# B&R Automation Studio project GAT (part 2)

### CutCamAut.axisfeature - 5PPC2200_AL14_000/mappMotion/CrossCutter/CutCamAut.axisfeature
```
Element CutterCamAutomat (Type=axisfeature)
  Type = CamAutomat
    CamAutomatType = ACOPOS
      CommonParameters:
        Master:
          ValueSource = SetPosition
            AxisReference = gAxisAppAxis_1
            MaxVelocity = 1000
          StartPosition = 0
          StartInterval = SpecifyValue
            Interval = 100
        AdvancedParameters:
          StartStateParameters:
            StartState = 0
            RelMasterStartPos = 0.0
          AdditiveAxes:
            AdditiveMasterValueSource = NotUsed
            AdditiveSlaveValueSource = NotUsed
          MasterStartPositionMode = NotEvaluatedAnew
          ControlSettings:
            CrossLeftBoundary = PositionLimitedHorizontal
            CamChangeImmediately = CurrentMasterMoveDir
          MessageSettings:
            ErrorsInStandby = NoErrorMessages
          TriggerAndLatch:
            Trigger1Delay = 0.0
            Trigger2Delay = 0.0
            SlaveLatchParID = 0
          EventParIDs
          StartIntervals
          Factors:
            SlaveFactorParID = 0
      States:
        State0 = Used
          Events:
            Event[0]:
              Type = MasterStartPosition
              Transition = Immediately
              SynchronousUpdate = Used
              NextState = 1
        State[1]  // Execute first cut
          Cam = Predefined
            PredefinedCam = OneToOne
          MasterFactor = 2000
          SlaveFactor = 2000
          CompensationMode = DistancesBetweenExitEntryPoints
            MasterDistance = 50
            SlaveDistance = 170
            AdvancedParameters = NotUsed
          AdvancedParameters:
            RepeatCounterInit = 0
            MasterValueSource = CommonMaster
          Events:
            Event[0]  // Stop cutting after next cut
              Type = Signal1FromPLC
              Transition = EndOfState
              SynchronousUpdate = Used
              NextState = 3
            Event[1]:
              Type = StateEnd
              Transition = EndOfState
              SynchronousUpdate = Used
              NextState = 2
        State[2]  // Execute cuts
          Cam = Predefined
            PredefinedCam = OneToOne
          MasterFactor = 2000
          SlaveFactor = 2000
          CompensationMode = DistancesBetweenCamCenterPoints
            MasterDistance = 100
            SlaveDistance = 360
            AdvancedParameters = NotUsed
          AdvancedParameters:
            RepeatCounterInit = 0
            MasterValueSource = CommonMaster
          Events:
            Event[0]  // Stop cutting after next cut
              Type = Signal1FromPLC
              Transition = EndOfState
              SynchronousUpdate = Used
              NextState = 3
            Event[1]:
              Type = StateEnd
              Transition = EndOfState
              SynchronousUpdate = Used
              NextState = 2
        State[3]  // decelerate and stop at home position
          Cam = Predefined
            PredefinedCam = ZeroPoint
          MasterFactor = 1000
          SlaveFactor = 0
          CompensationMode = DistancesBetweenCamCenterPoints
            MasterDistance = 50
            SlaveDistance = 180
            AdvancedParameters = NotUsed
          AdvancedParameters:
            RepeatCounterInit = 0
            MasterValueSource = CommonMaster
          Events:
            Event[0]:
              Type = StateEnd
              Transition = EndOfState
              SynchronousUpdate = Used
              NextState = 0
```

### CutVirt.purevaxcfg - 5PPC2200_AL14_000/mappMotion/CrossCutter/CutVirt.purevaxcfg
```
Element PureVAxCfg_CrossCutter (Type=purevaxcfg)
  TypeID = PureVAxConfig
  PureVAxis:
    AxisReference = gAxisCrossCutter
    Homing:
      Mode = Direct
        Position = 0.0
        ReferencePulse = NotUsed
      RestorePositionVariable
    JerkFilter = NotUsed
    AxisFeatures:
      FeatureRef[1] = CutterCamAutomat
```

### Alarm.mpalarmxcore - 5PPC2200_AL14_000/mappServices/AlarmX/Alarm.mpalarmxcore
```
Element gAlarmXMpLink (Type=mpalarmxcore)
  mapp.AlarmX.Core:
    BySeverity:
      [0]:
        Severity = 1..9
        [0] = Reaction
          Name = Info
      [1]:
        Severity = 10..19
        [0] = Reaction
          Name = Warning
      [2]:
        Severity = 20..29
        [0] = Reaction
          Name = Error
  mapp.AlarmX.Core.Configuration:
    [0]:
      Name = EmergencyStop_0
      Message = {$Alarms/EmergencyStop.0}
      Severity = 29
      Behavior = DiscreteValueMonitoring
        Monitoring:
          MonitoredPV = ::AlarmMgt:SafetyInputs.EmergencyStop[0]
          TriggerValues:
            [0] = 1
    [1]:
      Name = EmergencyStop_1
      Message = {$Alarms/EmergencyStop.1}
      Behavior = DiscreteValueMonitoring
        Monitoring:
          MonitoredPV = ::AlarmMgt:SafetyInputs.EmergencyStop[1]
          TriggerValues:
            [0] = 1
    [2]:
      Name = EmergencyStop_2
      Message = {$Alarms/EmergencyStop.2}
      Behavior = DiscreteValueMonitoring
        Monitoring:
          MonitoredPV = ::AlarmMgt:SafetyInputs.EmergencyStop[2]
          TriggerValues:
            [0] = 1
    [3]:
      Name = SafetyDoor_0
      Message = {$Alarms/SafetyDoor.0}
      Severity = 29
      Behavior = DiscreteValueMonitoring
        Monitoring:
          MonitoredPV = ::AlarmMgt:SafetyInputs.SafetyDoor[0]
          TriggerValues:
            [0] = 1
    [4]:
      Name = SafetyDoor_1
      Message = {$Alarms/SafetyDoor.1}
      Severity = 29
      Behavior = DiscreteValueMonitoring
        Monitoring:
          MonitoredPV = ::AlarmMgt:SafetyInputs.SafetyDoor[1]
          TriggerValues:
            [0] = 1
    [5]:
      Name = SafetyDoor_2
      Message = {$Alarms/SafetyDoor.2}
      Severity = 29
      Behavior = DiscreteValueMonitoring
        Monitoring:
          MonitoredPV = ::AlarmMgt:SafetyInputs.SafetyDoor[2]
          TriggerValues:
            [0] = 1
    [6]:
      Name = SafetyDoor_3
      Message = {$Alarms/SafetyDoor.3}
      Severity = 29
      Behavior = DiscreteValueMonitoring
        Monitoring:
          MonitoredPV = ::AlarmMgt:SafetyInputs.SafetyDoor[3]
          TriggerValues:
            [0] = 1
    [7]:
      Name = SafetyDoor_4
      Message = {$Alarms/SafetyDoor.4}
      Severity = 29
      Behavior = DiscreteValueMonitoring
        Monitoring:
          MonitoredPV = ::AlarmMgt:SafetyInputs.SafetyDoor[4]
          TriggerValues:
            [0] = 1
    [8]:
      Name = SafetyDoor_5
      Message = {$Alarms/SafetyDoor.5}
      Severity = 29
      Behavior = DiscreteValueMonitoring
        Monitoring:
          MonitoredPV = ::AlarmMgt:SafetyInputs.SafetyDoor[5]
          TriggerValues:
            [0] = 1
    [9]:
      Name = LevelMonitoringExample
      Message = {$Alarms/LevelMonitoringAlarmExample} {=$Alarms/{&LimitText}}
      Behavior = LevelMonitoring
        Monitoring:
          MonitoredPV = ::AlarmMgt:AlarmExamples.LevelMonitoring
          LowLimitEnable = Static
            Limit = 20
            LimitText = LevelMonitoringAlarmLowTextExample
            LowLowLimitEnable = Static
              Limit = 10
              LimitText = LevelMonitoringAlarmLowLowTextExample
          HighLimitEnable = Static
            Limit = 80
            LimitText = LevelMonitoringAlarmHighTextExample
            HighHighLimitEnable = Static
              Limit = 90
              LimitText = LevelMonitoringAlarmHighHighTextExample
    [10]:
      Name = DeviationMonitoringExample
      Message = {$Alarms/DeviationMonitoringAlarmExample} {&LimitText}
      Behavior = DeviationMonitoring
        Monitoring:
          MonitoredPV = ::AlarmMgt:AlarmExamples.DeviationMonitoring
          SetpointPV = ::AlarmMgt:AlarmExamples.DeviationMonitoringSetpoint
          LowLimitEnable = Static
            Limit = -5
            LimitText = Low limit exceeded
          HighLimitEnable = Static
            Limit = 5
            LimitText = High limit exceeded
    [11]:
      Name = RateOfChangeExample
      Message = {$Alarms/RateOfChangeAlarmExample}
      Behavior = RateOfChangeMonitoring
        Monitoring:
          MonitoredPV = ::AlarmMgt:AlarmExamples.RateOfChange
          HighLimitEnable = Static
            Limit = 5
            LimitText = High limit exceeded
    [12]:
      Name = SnippetExample
      Message = Show a snippet: {&snippet1}
      Behavior = DiscreteValueMonitoring
        Monitoring:
          MonitoredPV = ::AlarmMgt:AlarmExamples.SnippetValue
          TriggerValues:
            [0] = 50..100
    [13]:
      Name = MpAlarmXControlExample
      Message = {$Alarms/MpAlarmXControlExample}
      Severity = 20
      Behavior:
        Async = TRUE
    [14]:
      Name = Alarm0
      Message = {$Alarms/Alarm.0}
      Behavior = DiscreteValueMonitoring
        Monitoring:
          MonitoredPV = ::AlarmMgt:Alarms[0]
          InhibitPV = ::AlarmMgt:CommissioningModeActive
          TriggerValues:
            [0] = 1
    [15]:
      Name = Alarm1
      Message = {$Alarms/Alarm.1}
      Code = 1
      Behavior = DiscreteValueMonitoring
        Monitoring:
          MonitoredPV = ::AlarmMgt:Alarms[1]
          TriggerValues:
            [0] = 1
    [16]:
      Name = Alarm2
      Message = {$Alarms/Alarm.2}
      Code = 2
      Behavior = DiscreteValueMonitoring
        Monitoring:
          MonitoredPV = ::AlarmMgt:Alarms[2]
          TriggerValues:
            [0] = 1
    [17]:
      Name = Alarm3
      Message = {$Alarms/Alarm.3}
      Code = 3
      Behavior = DiscreteValueMonitoring
        Monitoring:
          MonitoredPV = ::AlarmMgt:Alarms[3]
          TriggerValues:
            [0] = 1
    [18]:
      Name = Alarm4
      Message = {$Alarms/Alarm.4}
      Code = 4
      Behavior = DiscreteValueMonitoring
        Monitoring:
          MonitoredPV = ::AlarmMgt:Alarms[4]
          TriggerValues:
            [0] = 1
    [19]:
      Name = Alarm5
      Message = {$Alarms/Alarm.5}
      Code = 5
      Behavior = DiscreteValueMonitoring
        Monitoring:
          MonitoredPV = ::AlarmMgt:Alarms[5]
          TriggerValues:
            [0] = 1
    [20]:
      Name = Alarm6
      Message = {$Alarms/Alarm.6}
      Code = 6
      Behavior = DiscreteValueMonitoring
        Monitoring:
          MonitoredPV = ::AlarmMgt:Alarms[6]
          TriggerValues:
            [0] = 1
    [21]:
      Name = Alarm7
      Message = {$Alarms/Alarm.7}
      Code = 7
      Behavior = DiscreteValueMonitoring
        Monitoring:
          MonitoredPV = ::AlarmMgt:Alarms[7]
          TriggerValues:
            [0] = 1
    [22]:
      Name = Alarm8
      Message = {$Alarms/Alarm.8}
      Code = 8
      Behavior = DiscreteValueMonitoring
        Monitoring:
          MonitoredPV = ::AlarmMgt:Alarms[8]
          TriggerValues:
            [0] = 1
    [23]:
      Name = Alarm9
      Message = {$Alarms/Alarm.9}
      Code = 9
      Behavior = DiscreteValueMonitoring
        Monitoring:
          MonitoredPV = ::AlarmMgt:Alarms[9]
          TriggerValues:
            [0] = 1
    [24]:
      Name = Alarm10
      Message = {$Alarms/Alarm.10}
      Code = 10
      Behavior = DiscreteValueMonitoring
        Monitoring:
          MonitoredPV = ::AlarmMgt:Alarms[10]
          TriggerValues:
            [0] = 1
    [25]:
      Name = Alarm11
      Message = {$Alarms/Alarm.11}
      Code = 11
      Behavior = DiscreteValueMonitoring
        Monitoring:
          MonitoredPV = ::AlarmMgt:Alarms[11]
          TriggerValues:
            [0] = 1
    [26]:
      Name = Alarm12
      Message = {$Alarms/Alarm.12}
      Code = 12
      Behavior = DiscreteValueMonitoring
        Monitoring:
          MonitoredPV = ::AlarmMgt:Alarms[12]
          TriggerValues:
            [0] = 1
    [27]:
      Name = Alarm13
      Message = {$Alarms/Alarm.13}
      Code = 13
      Behavior = DiscreteValueMonitoring
        Monitoring:
          MonitoredPV = ::AlarmMgt:Alarms[13]
          TriggerValues:
            [0] = 1
    [28]:
      Name = Alarm14
      Message = {$Alarms/Alarm.14}
      Code = 14
      Behavior = DiscreteValueMonitoring
        Monitoring:
          MonitoredPV = ::AlarmMgt:Alarms[14]
          TriggerValues:
            [0] = 1
    [29]:
      Name = Alarm15
      Message = {$Alarms/Alarm.15}
      Code = 15
      Behavior = DiscreteValueMonitoring
        Monitoring:
          MonitoredPV = ::AlarmMgt:Alarms[15]
          TriggerValues:
            [0] = 1
    [30]:
      Name = Alarm16
      Message = {$Alarms/Alarm.16}
      Code = 16
      Behavior = DiscreteValueMonitoring
        Monitoring:
          MonitoredPV = ::AlarmMgt:Alarms[16]
          TriggerValues:
            [0] = 1
    [31]:
      Name = Alarm17
      Message = {$Alarms/Alarm.17}
      Code = 17
      Behavior = DiscreteValueMonitoring
        Monitoring:
          MonitoredPV = ::AlarmMgt:Alarms[17]
          TriggerValues:
            [0] = 1
    [32]:
      Name = Alarm18
      Message = {$Alarms/Alarm.18}
      Code = 18
      Behavior = DiscreteValueMonitoring
        Monitoring:
          MonitoredPV = ::AlarmMgt:Alarms[18]
          TriggerValues:
            [0] = 1
    [33]:
      Name = Alarm19
      Message = {$Alarms/Alarm.19}
      Code = 19
      Behavior = DiscreteValueMonitoring
        Monitoring:
          MonitoredPV = ::AlarmMgt:Alarms[19]
          TriggerValues:
            [0] = 1
    [34]:
      Name = Alarm20
      Message = {$Alarms/Alarm.20}
      Behavior = DiscreteValueMonitoring
        Monitoring:
          MonitoredPV = ::AlarmMgt:Alarms[20]
          TriggerValues:
            [0] = 1
    [35]:
      Name = Alarm21
      Message = {$Alarms/Alarm.21}
      Code = 21
      Behavior = DiscreteValueMonitoring
        Monitoring:
          MonitoredPV = ::AlarmMgt:Alarms[21]
          TriggerValues:
            [0] = 1
    [36]:
      Name = Alarm22
      Message = {$Alarms/Alarm.22}
      Code = 22
      Behavior = DiscreteValueMonitoring
        Monitoring:
          MonitoredPV = ::AlarmMgt:Alarms[22]
          TriggerValues:
            [0] = 1
    [37]:
      Name = Alarm23
      Message = {$Alarms/Alarm.23}
      Code = 23
      Behavior = DiscreteValueMonitoring
        Monitoring:
          MonitoredPV = ::AlarmMgt:Alarms[23]
          TriggerValues:
            [0] = 1
    [38]:
      Name = Alarm24
      Message = {$Alarms/Alarm.24}
      Code = 24
      Behavior = DiscreteValueMonitoring
        Monitoring:
          MonitoredPV = ::AlarmMgt:Alarms[24]
          TriggerValues:
            [0] = 1
    [39]:
      Name = Alarm25
      Message = {$Alarms/Alarm.25}
      Code = 25
      Behavior = DiscreteValueMonitoring
        Monitoring:
          MonitoredPV = ::AlarmMgt:Alarms[25]
          TriggerValues:
            [0] = 1
    [40]:
      Name = Alarm26
      Message = {$Alarms/Alarm.26}
      Code = 26
      Behavior = DiscreteValueMonitoring
        Monitoring:
          MonitoredPV = ::AlarmMgt:Alarms[26]
          TriggerValues:
            [0] = 1
    [41]:
      Name = Alarm27
      Message = {$Alarms/Alarm.27}
      Code = 27
      Behavior = DiscreteValueMonitoring
        Monitoring:
          MonitoredPV = ::AlarmMgt:Alarms[27]
          TriggerValues:
            [0] = 1
    [42]:
      Name = Alarm28
      Message = {$Alarms/Alarm.28}
      Code = 28
      Behavior = DiscreteValueMonitoring
        Monitoring:
          MonitoredPV = ::AlarmMgt:Alarms[28]
          TriggerValues:
            [0] = 1
    [43]:
      Name = Alarm29
      Message = {$Alarms/Alarm.29}
      Code = 29
      Behavior = DiscreteValueMonitoring
        Monitoring:
          MonitoredPV = ::AlarmMgt:Alarms[29]
          TriggerValues:
            [0] = 1
    [44]:
      Name = Alarm30
      Message = {$Alarms/Alarm.30}
      Behavior = DiscreteValueMonitoring
        Monitoring:
          MonitoredPV = ::AlarmMgt:Alarms[30]
          TriggerValues:
            [0] = 1
    [45]:
      Name = Alarm31
      Message = {$Alarms/Alarm.31}
      Code = 31
      Behavior = DiscreteValueMonitoring
        Monitoring:
          MonitoredPV = ::AlarmMgt:Alarms[31]
          TriggerValues:
            [0] = 1
    [46]:
      Name = Alarm32
      Message = {$Alarms/Alarm.32}
      Code = 32
      Behavior = DiscreteValueMonitoring
        Monitoring:
          MonitoredPV = ::AlarmMgt:Alarms[32]
          TriggerValues:
            [0] = 1
    [47]:
      Name = Alarm33
      Message = {$Alarms/Alarm.33}
      Code = 33
      Behavior = DiscreteValueMonitoring
        Monitoring:
          MonitoredPV = ::AlarmMgt:Alarms[33]
          TriggerValues:
            [0] = 1
    [48]:
      Name = Alarm34
      Message = {$Alarms/Alarm.34}
      Code = 34
      Behavior = DiscreteValueMonitoring
        Monitoring:
          MonitoredPV = ::AlarmMgt:Alarms[34]
          TriggerValues:
            [0] = 1
    [49]:
      Name = Alarm35
      Message = {$Alarms/Alarm.35}
      Code = 35
      Behavior = DiscreteValueMonitoring
        Monitoring:
          MonitoredPV = ::AlarmMgt:Alarms[35]
          TriggerValues:
            [0] = 1
    [50]:
      Name = Alarm36
      Message = {$Alarms/Alarm.36}
      Code = 36
      Behavior = DiscreteValueMonitoring
        Monitoring:
          MonitoredPV = ::AlarmMgt:Alarms[36]
          TriggerValues:
            [0] = 1
    [51]:
      Name = Alarm37
      Message = {$Alarms/Alarm.37}
      Code = 37
      Behavior = DiscreteValueMonitoring
        Monitoring:
          MonitoredPV = ::AlarmMgt:Alarms[37]
          TriggerValues:
            [0] = 1
    [52]:
      Name = Alarm38
      Message = {$Alarms/Alarm.38}
      Code = 38
      Behavior = DiscreteValueMonitoring
        Monitoring:
          MonitoredPV = ::AlarmMgt:Alarms[38]
          TriggerValues:
            [0] = 1
    [53]:
      Name = Alarm39
      Message = {$Alarms/Alarm.39}
      Code = 39
      Behavior = DiscreteValueMonitoring
        Monitoring:
          MonitoredPV = ::AlarmMgt:Alarms[39]
          TriggerValues:
            [0] = 1
    [54]:
      Name = Alarm40
      Message = {$Alarms/Alarm.40}
      Behavior = DiscreteValueMonitoring
        Monitoring:
          MonitoredPV = ::AlarmMgt:Alarms[40]
          TriggerValues:
            [0] = 1
    [55]:
      Name = Alarm41
      Message = {$Alarms/Alarm.41}
      Code = 41
      Behavior = DiscreteValueMonitoring
        Monitoring:
          MonitoredPV = ::AlarmMgt:Alarms[41]
          TriggerValues:
            [0] = 1
    [56]:
      Name = Alarm42
      Message = {$Alarms/Alarm.42}
      Code = 42
      Behavior = DiscreteValueMonitoring
        Monitoring:
          MonitoredPV = ::AlarmMgt:Alarms[42]
          TriggerValues:
            [0] = 1
    [57]:
      Name = Alarm43
      Message = {$Alarms/Alarm.43}
      Code = 43
      Behavior = DiscreteValueMonitoring
        Monitoring:
          MonitoredPV = ::AlarmMgt:Alarms[43]
          TriggerValues:
            [0] = 1
    [58]:
      Name = Alarm44
      Message = {$Alarms/Alarm.44}
      Code = 44
      Behavior = DiscreteValueMonitoring
        Monitoring:
          MonitoredPV = ::AlarmMgt:Alarms[44]
          TriggerValues:
            [0] = 1
    [59]:
      Name = Alarm45
      Message = {$Alarms/Alarm.45}
      Code = 45
      Behavior = DiscreteValueMonitoring
        Monitoring:
          MonitoredPV = ::AlarmMgt:Alarms[45]
          TriggerValues:
            [0] = 1
    [60]:
      Name = Alarm46
      Message = {$Alarms/Alarm.46}
      Code = 46
      Behavior = DiscreteValueMonitoring
        Monitoring:
          MonitoredPV = ::AlarmMgt:Alarms[46]
          TriggerValues:
            [0] = 1
    [61]:
      Name = Alarm47
      Message = {$Alarms/Alarm.47}
      Code = 47
      Behavior = DiscreteValueMonitoring
        Monitoring:
          MonitoredPV = ::AlarmMgt:Alarms[47]
          TriggerValues:
            [0] = 1
    [62]:
      Name = Alarm48
      Message = {$Alarms/Alarm.48}
      Code = 48
      Behavior = DiscreteValueMonitoring
        Monitoring:
          MonitoredPV = ::AlarmMgt:Alarms[48]
          TriggerValues:
            [0] = 1
    [63]:
      Name = Alarm49
      Message = {$Alarms/Alarm.49}
      Code = 49
      Behavior = DiscreteValueMonitoring
        Monitoring:
          MonitoredPV = ::AlarmMgt:Alarms[49]
          TriggerValues:
            [0] = 1
    [64]:
      Name = Alarm50
      Message = {$Alarms/Alarm.50}
      Behavior = DiscreteValueMonitoring
        Monitoring:
          MonitoredPV = ::AlarmMgt:Alarms[50]
          TriggerValues:
            [0] = 1
    [65]:
      Name = Alarm51
      Message = {$Alarms/Alarm.51}
      Code = 51
      Behavior = DiscreteValueMonitoring
        Monitoring:
          MonitoredPV = ::AlarmMgt:Alarms[51]
          TriggerValues:
            [0] = 1
    [66]:
      Name = Alarm52
      Message = {$Alarms/Alarm.52}
      Code = 52
      Behavior = DiscreteValueMonitoring
        Monitoring:
          MonitoredPV = ::AlarmMgt:Alarms[52]
          TriggerValues:
            [0] = 1
    [67]:
      Name = Alarm53
      Message = {$Alarms/Alarm.53}
      Code = 53
      Behavior = DiscreteValueMonitoring
        Monitoring:
          MonitoredPV = ::AlarmMgt:Alarms[53]
          TriggerValues:
            [0] = 1
    [68]:
      Name = Alarm54
      Message = {$Alarms/Alarm.54}
      Code = 54
      Behavior = DiscreteValueMonitoring
        Monitoring:
          MonitoredPV = ::AlarmMgt:Alarms[54]
          TriggerValues:
            [0] = 1
    [69]:
      Name = Alarm55
      Message = {$Alarms/Alarm.55}
      Code = 55
      Behavior = DiscreteValueMonitoring
        Monitoring:
          MonitoredPV = ::AlarmMgt:Alarms[55]
          TriggerValues:
            [0] = 1
    [70]:
      Name = Alarm56
      Message = {$Alarms/Alarm.56}
      Code = 56
      Behavior = DiscreteValueMonitoring
        Monitoring:
          MonitoredPV = ::AlarmMgt:Alarms[56]
          TriggerValues:
            [0] = 1
    [71]:
      Name = Alarm57
      Message = {$Alarms/Alarm.57}
      Code = 57
      Behavior = DiscreteValueMonitoring
        Monitoring:
          MonitoredPV = ::AlarmMgt:Alarms[57]
          TriggerValues:
            [0] = 1
    [72]:
      Name = Alarm58
      Message = {$Alarms/Alarm.58}
      Code = 58
      Behavior = DiscreteValueMonitoring
        Monitoring:
          MonitoredPV = ::AlarmMgt:Alarms[58]
          TriggerValues:
            [0] = 1
    [73]:
      Name = Alarm59
      Message = {$Alarms/Alarm.59}
      Code = 59
      Behavior = DiscreteValueMonitoring
        Monitoring:
          MonitoredPV = ::AlarmMgt:Alarms[59]
          TriggerValues:
            [0] = 1
    [74]:
      Name = Alarm60
      Message = {$Alarms/Alarm.60}
      Behavior = DiscreteValueMonitoring
        Monitoring:
          MonitoredPV = ::AlarmMgt:Alarms[60]
          TriggerValues:
            [0] = 1
    [75]:
      Name = Alarm61
      Message = {$Alarms/Alarm.61}
      Code = 61
      Behavior = DiscreteValueMonitoring
        Monitoring:
          MonitoredPV = ::AlarmMgt:Alarms[61]
          TriggerValues:
            [0] = 1
    [76]:
      Name = Alarm62
      Message = {$Alarms/Alarm.62}
      Code = 62
      Behavior = DiscreteValueMonitoring
        Monitoring:
          MonitoredPV = ::AlarmMgt:Alarms[62]
          TriggerValues:
            [0] = 1
    [77]:
      Name = Alarm63
      Message = {$Alarms/Alarm.63}
      Code = 63
      Behavior = DiscreteValueMonitoring
        Monitoring:
          MonitoredPV = ::AlarmMgt:Alarms[63]
          TriggerValues:
            [0] = 1
    [78]:
      Name = Alarm64
      Message = {$Alarms/Alarm.64}
      Code = 64
      Behavior = DiscreteValueMonitoring
        Monitoring:
          MonitoredPV = ::AlarmMgt:Alarms[64]
          TriggerValues:
            [0] = 1
    [79]:
      Name = Alarm65
      Message = {$Alarms/Alarm.65}
      Code = 65
      Behavior = DiscreteValueMonitoring
        Monitoring:
          MonitoredPV = ::AlarmMgt:Alarms[65]
          TriggerValues:
            [0] = 1
    [80]:
      Name = Alarm66
      Message = {$Alarms/Alarm.66}
      Code = 66
      Behavior = DiscreteValueMonitoring
        Monitoring:
          MonitoredPV = ::AlarmMgt:Alarms[66]
          TriggerValues:
            [0] = 1
    [81]:
      Name = Alarm67
      Message = {$Alarms/Alarm.67}
      Code = 67
      Behavior = DiscreteValueMonitoring
        Monitoring:
          MonitoredPV = ::AlarmMgt:Alarms[67]
          TriggerValues:
            [0] = 1
    [82]:
      Name = Alarm68
      Message = {$Alarms/Alarm.68}
      Code = 68
      Behavior = DiscreteValueMonitoring
        Monitoring:
          MonitoredPV = ::AlarmMgt:Alarms[68]
          TriggerValues:
            [0] = 1
    [83]:
      Name = Alarm69
      Message = {$Alarms/Alarm.69}
      Code = 69
      Behavior = DiscreteValueMonitoring
        Monitoring:
          MonitoredPV = ::AlarmMgt:Alarms[69]
          TriggerValues:
            [0] = 1
    [84]:
      Name = Alarm70
      Message = {$Alarms/Alarm.70}
      Behavior = DiscreteValueMonitoring
        Monitoring:
          MonitoredPV = ::AlarmMgt:Alarms[70]
          TriggerValues:
            [0] = 1
    [85]:
      Name = Alarm71
      Message = {$Alarms/Alarm.71}
      Code = 71
      Behavior = DiscreteValueMonitoring
        Monitoring:
          MonitoredPV = ::AlarmMgt:Alarms[71]
          TriggerValues:
            [0] = 1
    [86]:
      Name = Alarm72
      Message = {$Alarms/Alarm.72}
      Code = 72
      Behavior = DiscreteValueMonitoring
        Monitoring:
          MonitoredPV = ::AlarmMgt:Alarms[72]
          TriggerValues:
            [0] = 1
    [87]:
      Name = Alarm73
      Message = {$Alarms/Alarm.73}
      Code = 73
      Behavior = DiscreteValueMonitoring
        Monitoring:
          MonitoredPV = ::AlarmMgt:Alarms[73]
          TriggerValues:
            [0] = 1
    [88]:
      Name = Alarm74
      Message = {$Alarms/Alarm.74}
      Code = 74
      Behavior = DiscreteValueMonitoring
        Monitoring:
          MonitoredPV = ::AlarmMgt:Alarms[74]
          TriggerValues:
            [0] = 1
    [89]:
      Name = Alarm75
      Message = {$Alarms/Alarm.75}
      Code = 75
      Behavior = DiscreteValueMonitoring
        Monitoring:
          MonitoredPV = ::AlarmMgt:Alarms[75]
          TriggerValues:
            [0] = 1
    [90]:
      Name = Alarm76
      Message = {$Alarms/Alarm.76}
      Code = 76
      Behavior = DiscreteValueMonitoring
        Monitoring:
          MonitoredPV = ::AlarmMgt:Alarms[76]
          TriggerValues:
            [0] = 1
    [91]:
      Name = Alarm77
      Message = {$Alarms/Alarm.77}
      Code = 77
      Behavior = DiscreteValueMonitoring
        Monitoring:
          MonitoredPV = ::AlarmMgt:Alarms[77]
          TriggerValues:
            [0] = 1
    [92]:
      Name = Alarm78
      Message = {$Alarms/Alarm.78}
      Code = 78
      Behavior = DiscreteValueMonitoring
        Monitoring:
          MonitoredPV = ::AlarmMgt:Alarms[78]
          TriggerValues:
            [0] = 1
    [93]:
      Name = Alarm79
      Message = {$Alarms/Alarm.79}
      Code = 79
      Behavior = DiscreteValueMonitoring
        Monitoring:
          MonitoredPV = ::AlarmMgt:Alarms[79]
          TriggerValues:
            [0] = 1
    [94]:
      Name = Alarm80
      Message = {$Alarms/Alarm.80}
      Behavior = DiscreteValueMonitoring
        Monitoring:
          MonitoredPV = ::AlarmMgt:Alarms[80]
          TriggerValues:
            [0] = 1
    [95]:
      Name = Alarm81
      Message = {$Alarms/Alarm.81}
      Code = 81
      Behavior = DiscreteValueMonitoring
        Monitoring:
          MonitoredPV = ::AlarmMgt:Alarms[81]
          TriggerValues:
            [0] = 1
    [96]:
      Name = Alarm82
      Message = {$Alarms/Alarm.82}
      Code = 82
      Behavior = DiscreteValueMonitoring
        Monitoring:
          MonitoredPV = ::AlarmMgt:Alarms[82]
          TriggerValues:
            [0] = 1
    [97]:
      Name = Alarm83
      Message = {$Alarms/Alarm.83}
      Code = 83
      Behavior = DiscreteValueMonitoring
        Monitoring:
          MonitoredPV = ::AlarmMgt:Alarms[83]
          TriggerValues:
            [0] = 1
    [98]:
      Name = Alarm84
      Message = {$Alarms/Alarm.84}
      Code = 84
      Behavior = DiscreteValueMonitoring
        Monitoring:
          MonitoredPV = ::AlarmMgt:Alarms[84]
          TriggerValues:
            [0] = 1
    [99]:
      Name = Alarm85
      Message = {$Alarms/Alarm.85}
      Code = 85
      Behavior = DiscreteValueMonitoring
        Monitoring:
          MonitoredPV = ::AlarmMgt:Alarms[85]
          TriggerValues:
            [0] = 1
    [100]:
      Name = Alarm86
      Message = {$Alarms/Alarm.86}
      Code = 86
      Behavior = DiscreteValueMonitoring
        Monitoring:
          MonitoredPV = ::AlarmMgt:Alarms[86]
          TriggerValues:
            [0] = 1
    [101]:
      Name = Alarm87
      Message = {$Alarms/Alarm.87}
      Code = 87
      Behavior = DiscreteValueMonitoring
        Monitoring:
          MonitoredPV = ::AlarmMgt:Alarms[87]
          TriggerValues:
            [0] = 1
    [102]:
      Name = Alarm88
      Message = {$Alarms/Alarm.88}
      Code = 88
      Behavior = DiscreteValueMonitoring
        Monitoring:
          MonitoredPV = ::AlarmMgt:Alarms[88]
          TriggerValues:
            [0] = 1
    [103]:
      Name = Alarm89
      Message = {$Alarms/Alarm.89}
      Code = 89
      Behavior = DiscreteValueMonitoring
        Monitoring:
          MonitoredPV = ::AlarmMgt:Alarms[89]
          TriggerValues:
            [0] = 1
    [104]:
      Name = Alarm90
      Message = {$Alarms/Alarm.90}
      Behavior = DiscreteValueMonitoring
        Monitoring:
          MonitoredPV = ::AlarmMgt:Alarms[90]
          TriggerValues:
            [0] = 1
    [105]:
      Name = Alarm91
      Message = {$Alarms/Alarm.91}
      Code = 91
      Behavior = DiscreteValueMonitoring
        Monitoring:
          MonitoredPV = ::AlarmMgt:Alarms[91]
          TriggerValues:
            [0] = 1
    [106]:
      Name = Alarm92
      Message = {$Alarms/Alarm.92}
      Code = 92
      Behavior = DiscreteValueMonitoring
        Monitoring:
          MonitoredPV = ::AlarmMgt:Alarms[92]
          TriggerValues:
            [0] = 1
    [107]:
      Name = Alarm93
      Message = {$Alarms/Alarm.93}
      Code = 93
      Behavior = DiscreteValueMonitoring
        Monitoring:
          MonitoredPV = ::AlarmMgt:Alarms[93]
          TriggerValues:
            [0] = 1
    [108]:
      Name = Alarm94
      Message = {$Alarms/Alarm.94}
      Code = 94
      Behavior = DiscreteValueMonitoring
        Monitoring:
          MonitoredPV = ::AlarmMgt:Alarms[94]
          TriggerValues:
            [0] = 1
    [109]:
      Name = Alarm95
      Message = {$Alarms/Alarm.95}
      Code = 95
      Behavior = DiscreteValueMonitoring
        Monitoring:
          MonitoredPV = ::AlarmMgt:Alarms[95]
          TriggerValues:
            [0] = 1
    [110]:
      Name = Alarm96
      Message = {$Alarms/Alarm.96}
      Code = 96
      Behavior = DiscreteValueMonitoring
        Monitoring:
          MonitoredPV = ::AlarmMgt:Alarms[96]
          TriggerValues:
            [0] = 1
    [111]:
      Name = Alarm97
      Message = {$Alarms/Alarm.97}
      Code = 97
      Behavior = DiscreteValueMonitoring
        Monitoring:
          MonitoredPV = ::AlarmMgt:Alarms[97]
          TriggerValues:
            [0] = 1
    [112]:
      Name = Alarm98
      Message = {$Alarms/Alarm.98}
      Code = 98
      Behavior = DiscreteValueMonitoring
        Monitoring:
          MonitoredPV = ::AlarmMgt:Alarms[98]
          TriggerValues:
            [0] = 1
    [113]:
      Name = Alarm99
      Message = {$Alarms/Alarm.99}
      Code = 99
      Behavior = DiscreteValueMonitoring
        Monitoring:
          MonitoredPV = ::AlarmMgt:Alarms[99]
          TriggerValues:
            [0] = 1
  mapp.AlarmX.Core.Snippets:
    AutoDetect = 1
    [0]:
      Key = snippet1
      Value:
        PV = ::AlarmMgt:AlarmExamples.SnippetValue
  mapp.AlarmX.Core.Queries:
    [0]:
      Name = ActiveAlarms
      Update = ::AlarmMgt:AlarmQuery.ActiveAlarmUpdateCount
      Source:
        SELECT:
          [0]:
            PV = ::AlarmMgt:AlarmQuery.Alarms[].Name
          [1]:
            Column = Message
            PV = ::AlarmMgt:AlarmQuery.Alarms[].Message
          [2]:
            Column = Code
            PV = ::AlarmMgt:AlarmQuery.Alarms[].Code
          [3]:
            Column = Severity
            PV = ::AlarmMgt:AlarmQuery.Alarms[].Severity
          [4]:
            Column = Scope
            PV = ::AlarmMgt:AlarmQuery.Alarms[].Scope
          [5]:
            Column = TimeStamp
            PV = ::AlarmMgt:AlarmQuery.Alarms[].TimeStamp
          [6]:
            Column = AdditionalInformation1
            PV = ::AlarmMgt:AlarmQuery.Alarms[].AdditionalInfo
          [7]:
            Column = StateActive
            PV = ::AlarmMgt:AlarmQuery.Alarms[].Active
          [8]:
            Column = StateAcknowledged
            PV = ::AlarmMgt:AlarmQuery.Alarms[].Acknowledged
```

### AlarmX.mpalarmxcore - 5PPC2200_AL14_000/mappServices/AlarmX/AlarmX.mpalarmxcore
```
Element gMpLinkAlarmXCore (Type=mpalarmxcore)
  mapp.AlarmX.Core:
    BySeverity:
      [0]:
        Severity = 1..9
        [0] = Reaction
          Name = Info
      [1]:
        Severity = 10..19
        [0] = Reaction
          Name = Warning
      [2]:
        Severity = 20..29
        [0] = Reaction
          Name = Error
  mapp.AlarmX.Core.Configuration:
    [0]:
      Name = EmergencyStop_0
      Message = {$Alarms/EmergencyStop.0}
      Severity = 29
      Behavior = DiscreteValueMonitoring
        Monitoring:
          MonitoredPV = ::AlarmMgt:SafetyInputs.EmergencyStop[0]
          TriggerValues:
            [0] = 1
    [1]:
      Name = EmergencyStop_1
      Message = {$Alarms/EmergencyStop.1}
      Behavior = DiscreteValueMonitoring
        Monitoring:
          MonitoredPV = ::AlarmMgt:SafetyInputs.EmergencyStop[1]
          TriggerValues:
            [0] = 1
    [2]:
      Name = EmergencyStop_2
      Message = {$Alarms/EmergencyStop.2}
      Behavior = DiscreteValueMonitoring
        Monitoring:
          MonitoredPV = ::AlarmMgt:SafetyInputs.EmergencyStop[2]
          TriggerValues:
            [0] = 1
    [3]:
      Name = SafetyDoor_0
      Message = {$Alarms/SafetyDoor.0}
      Severity = 29
      Behavior = DiscreteValueMonitoring
        Monitoring:
          MonitoredPV = ::AlarmMgt:SafetyInputs.SafetyDoor[0]
          TriggerValues:
            [0] = 1
    [4]:
      Name = SafetyDoor_1
      Message = {$Alarms/SafetyDoor.1}
      Severity = 29
      Behavior = DiscreteValueMonitoring
        Monitoring:
          MonitoredPV = ::AlarmMgt:SafetyInputs.SafetyDoor[1]
          TriggerValues:
            [0] = 1
    [5]:
      Name = SafetyDoor_2
      Message = {$Alarms/SafetyDoor.2}
      Severity = 29
      Behavior = DiscreteValueMonitoring
        Monitoring:
          MonitoredPV = ::AlarmMgt:SafetyInputs.SafetyDoor[2]
          TriggerValues:
            [0] = 1
    [6]:
      Name = SafetyDoor_3
      Message = {$Alarms/SafetyDoor.3}
      Severity = 29
      Behavior = DiscreteValueMonitoring
        Monitoring:
          MonitoredPV = ::AlarmMgt:SafetyInputs.SafetyDoor[3]
          TriggerValues:
            [0] = 1
    [7]:
      Name = SafetyDoor_4
      Message = {$Alarms/SafetyDoor.4}
      Severity = 29
      Behavior = DiscreteValueMonitoring
        Monitoring:
          MonitoredPV = ::AlarmMgt:SafetyInputs.SafetyDoor[4]
          TriggerValues:
            [0] = 1
    [8]:
      Name = SafetyDoor_5
      Message = {$Alarms/SafetyDoor.5}
      Severity = 29
      Behavior = DiscreteValueMonitoring
        Monitoring:
          MonitoredPV = ::AlarmMgt:SafetyInputs.SafetyDoor[5]
          TriggerValues:
            [0] = 1
    [9]:
      Name = LevelMonitoringExample
      Message = {$Alarms/LevelMonitoringAlarmExample} {=$Alarms/{&LimitText}}
      Behavior = LevelMonitoring
        Monitoring:
          MonitoredPV = ::AlarmMgt:AlarmExamples.LevelMonitoring
          LowLimitEnable = Static
            Limit = 20
            LimitText = LevelMonitoringAlarmLowTextExample
            LowLowLimitEnable = Static
              Limit = 10
              LimitText = LevelMonitoringAlarmLowLowTextExample
          HighLimitEnable = Static
            Limit = 80
            LimitText = LevelMonitoringAlarmHighTextExample
            HighHighLimitEnable = Static
              Limit = 90
              LimitText = LevelMonitoringAlarmHighHighTextExample
    [10]:
      Name = DeviationMonitoringExample
      Message = {$Alarms/DeviationMonitoringAlarmExample} {&LimitText}
      Behavior = DeviationMonitoring
        Monitoring:
          MonitoredPV = ::AlarmMgt:AlarmExamples.DeviationMonitoring
          SetpointPV = ::AlarmMgt:AlarmExamples.DeviationMonitoringSetpoint
          LowLimitEnable = Static
            Limit = -5
            LimitText = Low limit exceeded
          HighLimitEnable = Static
            Limit = 5
            LimitText = High limit exceeded
    [11]:
      Name = RateOfChangeExample
      Message = {$Alarms/RateOfChangeAlarmExample}
      Behavior = RateOfChangeMonitoring
        Monitoring:
          MonitoredPV = ::AlarmMgt:AlarmExamples.RateOfChange
          HighLimitEnable = Static
            Limit = 5
            LimitText = High limit exceeded
    [12]:
      Name = SnippetExample
      Message = Show a snippet: {&snippet1}
      Behavior = DiscreteValueMonitoring
        Monitoring:
          MonitoredPV = ::AlarmMgt:AlarmExamples.SnippetValue
          TriggerValues:
            [0] = 50..100
    [13]:
      Name = MpAlarmXControlExample
      Message = {$Alarms/MpAlarmXControlExample}
      Severity = 20
      Behavior:
        Async = TRUE
    [14]:
      Name = Alarm0
      Message = {$Alarms/Alarm.0}
      Behavior = DiscreteValueMonitoring
        Monitoring:
          MonitoredPV = ::AlarmMgt:Alarms[0]
          InhibitPV = ::AlarmMgt:CommissioningModeActive
          TriggerValues:
            [0] = 1
    [15]:
      Name = Alarm1
      Message = {$Alarms/Alarm.1}
      Code = 1
      Behavior = DiscreteValueMonitoring
        Monitoring:
          MonitoredPV = ::AlarmMgt:Alarms[1]
          TriggerValues:
            [0] = 1
    [16]:
      Name = Alarm2
      Message = {$Alarms/Alarm.2}
      Code = 2
      Behavior = DiscreteValueMonitoring
        Monitoring:
          MonitoredPV = ::AlarmMgt:Alarms[2]
          TriggerValues:
            [0] = 1
    [17]:
      Name = Alarm3
      Message = {$Alarms/Alarm.3}
      Code = 3
      Behavior = DiscreteValueMonitoring
        Monitoring:
          MonitoredPV = ::AlarmMgt:Alarms[3]
          TriggerValues:
            [0] = 1
    [18]:
      Name = Alarm4
      Message = {$Alarms/Alarm.4}
      Code = 4
      Behavior = DiscreteValueMonitoring
        Monitoring:
          MonitoredPV = ::AlarmMgt:Alarms[4]
          TriggerValues:
            [0] = 1
    [19]:
      Name = Alarm5
      Message = {$Alarms/Alarm.5}
      Code = 5
      Behavior = DiscreteValueMonitoring
        Monitoring:
          MonitoredPV = ::AlarmMgt:Alarms[5]
          TriggerValues:
            [0] = 1
    [20]:
      Name = Alarm6
      Message = {$Alarms/Alarm.6}
      Code = 6
      Behavior = DiscreteValueMonitoring
        Monitoring:
          MonitoredPV = ::AlarmMgt:Alarms[6]
          TriggerValues:
            [0] = 1
    [21]:
      Name = Alarm7
      Message = {$Alarms/Alarm.7}
      Code = 7
      Behavior = DiscreteValueMonitoring
        Monitoring:
          MonitoredPV = ::AlarmMgt:Alarms[7]
          TriggerValues:
            [0] = 1
    [22]:
      Name = Alarm8
      Message = {$Alarms/Alarm.8}
      Code = 8
      Behavior = DiscreteValueMonitoring
        Monitoring:
          MonitoredPV = ::AlarmMgt:Alarms[8]
          TriggerValues:
            [0] = 1
    [23]:
      Name = Alarm9
      Message = {$Alarms/Alarm.9}
      Code = 9
      Behavior = DiscreteValueMonitoring
        Monitoring:
          MonitoredPV = ::AlarmMgt:Alarms[9]
          TriggerValues:
            [0] = 1
    [24]:
      Name = Alarm10
      Message = {$Alarms/Alarm.10}
      Code = 10
      Behavior = DiscreteValueMonitoring
        Monitoring:
          MonitoredPV = ::AlarmMgt:Alarms[10]
          TriggerValues:
            [0] = 1
    [25]:
      Name = Alarm11
      Message = {$Alarms/Alarm.11}
      Code = 11
      Behavior = DiscreteValueMonitoring
        Monitoring:
          MonitoredPV = ::AlarmMgt:Alarms[11]
          TriggerValues:
            [0] = 1
    [26]:
      Name = Alarm12
      Message = {$Alarms/Alarm.12}
      Code = 12
      Behavior = DiscreteValueMonitoring
        Monitoring:
          MonitoredPV = ::AlarmMgt:Alarms[12]
          TriggerValues:
            [0] = 1
    [27]:
      Name = Alarm13
      Message = {$Alarms/Alarm.13}
      Code = 13
      Behavior = DiscreteValueMonitoring
        Monitoring:
          MonitoredPV = ::AlarmMgt:Alarms[13]
          TriggerValues:
            [0] = 1
    [28]:
      Name = Alarm14
      Message = {$Alarms/Alarm.14}
      Code = 14
      Behavior = DiscreteValueMonitoring
        Monitoring:
          MonitoredPV = ::AlarmMgt:Alarms[14]
          TriggerValues:
            [0] = 1
    [29]:
      Name = Alarm15
      Message = {$Alarms/Alarm.15}
      Code = 15
      Behavior = DiscreteValueMonitoring
        Monitoring:
          MonitoredPV = ::AlarmMgt:Alarms[15]
          TriggerValues:
            [0] = 1
    [30]:
      Name = Alarm16
      Message = {$Alarms/Alarm.16}
      Code = 16
      Behavior = DiscreteValueMonitoring
        Monitoring:
          MonitoredPV = ::AlarmMgt:Alarms[16]
          TriggerValues:
            [0] = 1
    [31]:
      Name = Alarm17
      Message = {$Alarms/Alarm.17}
      Code = 17
      Behavior = DiscreteValueMonitoring
        Monitoring:
          MonitoredPV = ::AlarmMgt:Alarms[17]
          TriggerValues:
            [0] = 1
    [32]:
      Name = Alarm18
      Message = {$Alarms/Alarm.18}
      Code = 18
      Behavior = DiscreteValueMonitoring
        Monitoring:
          MonitoredPV = ::AlarmMgt:Alarms[18]
          TriggerValues:
            [0] = 1
    [33]:
      Name = Alarm19
      Message = {$Alarms/Alarm.19}
      Code = 19
      Behavior = DiscreteValueMonitoring
        Monitoring:
          MonitoredPV = ::AlarmMgt:Alarms[19]
          TriggerValues:
            [0] = 1
    [34]:
      Name = Alarm20
      Message = {$Alarms/Alarm.20}
      Behavior = DiscreteValueMonitoring
        Monitoring:
          MonitoredPV = ::AlarmMgt:Alarms[20]
          TriggerValues:
            [0] = 1
    [35]:
      Name = Alarm21
      Message = {$Alarms/Alarm.21}
      Code = 21
      Behavior = DiscreteValueMonitoring
        Monitoring:
          MonitoredPV = ::AlarmMgt:Alarms[21]
          TriggerValues:
            [0] = 1
    [36]:
      Name = Alarm22
      Message = {$Alarms/Alarm.22}
      Code = 22
      Behavior = DiscreteValueMonitoring
        Monitoring:
          MonitoredPV = ::AlarmMgt:Alarms[22]
          TriggerValues:
            [0] = 1
    [37]:
      Name = Alarm23
      Message = {$Alarms/Alarm.23}
      Code = 23
      Behavior = DiscreteValueMonitoring
        Monitoring:
          MonitoredPV = ::AlarmMgt:Alarms[23]
          TriggerValues:
            [0] = 1
    [38]:
      Name = Alarm24
      Message = {$Alarms/Alarm.24}
      Code = 24
      Behavior = DiscreteValueMonitoring
        Monitoring:
          MonitoredPV = ::AlarmMgt:Alarms[24]
          TriggerValues:
            [0] = 1
    [39]:
      Name = Alarm25
      Message = {$Alarms/Alarm.25}
      Code = 25
      Behavior = DiscreteValueMonitoring
        Monitoring:
          MonitoredPV = ::AlarmMgt:Alarms[25]
          TriggerValues:
            [0] = 1
    [40]:
      Name = Alarm26
      Message = {$Alarms/Alarm.26}
      Code = 26
      Behavior = DiscreteValueMonitoring
        Monitoring:
          MonitoredPV = ::AlarmMgt:Alarms[26]
          TriggerValues:
            [0] = 1
    [41]:
      Name = Alarm27
      Message = {$Alarms/Alarm.27}
      Code = 27
      Behavior = DiscreteValueMonitoring
        Monitoring:
          MonitoredPV = ::AlarmMgt:Alarms[27]
          TriggerValues:
            [0] = 1
    [42]:
      Name = Alarm28
      Message = {$Alarms/Alarm.28}
      Code = 28
      Behavior = DiscreteValueMonitoring
        Monitoring:
          MonitoredPV = ::AlarmMgt:Alarms[28]
          TriggerValues:
            [0] = 1
    [43]:
      Name = Alarm29
      Message = {$Alarms/Alarm.29}
      Code = 29
      Behavior = DiscreteValueMonitoring
        Monitoring:
          MonitoredPV = ::AlarmMgt:Alarms[29]
          TriggerValues:
            [0] = 1
    [44]:
      Name = Alarm30
      Message = {$Alarms/Alarm.30}
      Behavior = DiscreteValueMonitoring
        Monitoring:
          MonitoredPV = ::AlarmMgt:Alarms[30]
          TriggerValues:
            [0] = 1
    [45]:
      Name = Alarm31
      Message = {$Alarms/Alarm.31}
      Code = 31
      Behavior = DiscreteValueMonitoring
        Monitoring:
          MonitoredPV = ::AlarmMgt:Alarms[31]
          TriggerValues:
            [0] = 1
    [46]:
      Name = Alarm32
      Message = {$Alarms/Alarm.32}
      Code = 32
      Behavior = DiscreteValueMonitoring
        Monitoring:
          MonitoredPV = ::AlarmMgt:Alarms[32]
          TriggerValues:
            [0] = 1
    [47]:
      Name = Alarm33
      Message = {$Alarms/Alarm.33}
      Code = 33
      Behavior = DiscreteValueMonitoring
        Monitoring:
          MonitoredPV = ::AlarmMgt:Alarms[33]
          TriggerValues:
            [0] = 1
    [48]:
      Name = Alarm34
      Message = {$Alarms/Alarm.34}
      Code = 34
      Behavior = DiscreteValueMonitoring
        Monitoring:
          MonitoredPV = ::AlarmMgt:Alarms[34]
          TriggerValues:
            [0] = 1
    [49]:
      Name = Alarm35
      Message = {$Alarms/Alarm.35}
      Code = 35
      Behavior = DiscreteValueMonitoring
        Monitoring:
          MonitoredPV = ::AlarmMgt:Alarms[35]
          TriggerValues:
            [0] = 1
    [50]:
      Name = Alarm36
      Message = {$Alarms/Alarm.36}
      Code = 36
      Behavior = DiscreteValueMonitoring
        Monitoring:
          MonitoredPV = ::AlarmMgt:Alarms[36]
          TriggerValues:
            [0] = 1
    [51]:
      Name = Alarm37
      Message = {$Alarms/Alarm.37}
      Code = 37
      Behavior = DiscreteValueMonitoring
        Monitoring:
          MonitoredPV = ::AlarmMgt:Alarms[37]
          TriggerValues:
            [0] = 1
    [52]:
      Name = Alarm38
      Message = {$Alarms/Alarm.38}
      Code = 38
      Behavior = DiscreteValueMonitoring
        Monitoring:
          MonitoredPV = ::AlarmMgt:Alarms[38]
          TriggerValues:
            [0] = 1
    [53]:
      Name = Alarm39
      Message = {$Alarms/Alarm.39}
      Code = 39
      Behavior = DiscreteValueMonitoring
        Monitoring:
          MonitoredPV = ::AlarmMgt:Alarms[39]
          TriggerValues:
            [0] = 1
    [54]:
      Name = Alarm40
      Message = {$Alarms/Alarm.40}
      Behavior = DiscreteValueMonitoring
        Monitoring:
          MonitoredPV = ::AlarmMgt:Alarms[40]
          TriggerValues:
            [0] = 1
    [55]:
      Name = Alarm41
      Message = {$Alarms/Alarm.41}
      Code = 41
      Behavior = DiscreteValueMonitoring
        Monitoring:
          MonitoredPV = ::AlarmMgt:Alarms[41]
          TriggerValues:
            [0] = 1
    [56]:
      Name = Alarm42
      Message = {$Alarms/Alarm.42}
      Code = 42
      Behavior = DiscreteValueMonitoring
        Monitoring:
          MonitoredPV = ::AlarmMgt:Alarms[42]
          TriggerValues:
            [0] = 1
    [57]:
      Name = Alarm43
      Message = {$Alarms/Alarm.43}
      Code = 43
      Behavior = DiscreteValueMonitoring
        Monitoring:
          MonitoredPV = ::AlarmMgt:Alarms[43]
          TriggerValues:
            [0] = 1
    [58]:
      Name = Alarm44
      Message = {$Alarms/Alarm.44}
      Code = 44
      Behavior = DiscreteValueMonitoring
        Monitoring:
          MonitoredPV = ::AlarmMgt:Alarms[44]
          TriggerValues:
            [0] = 1
    [59]:
      Name = Alarm45
      Message = {$Alarms/Alarm.45}
      Code = 45
      Behavior = DiscreteValueMonitoring
        Monitoring:
          MonitoredPV = ::AlarmMgt:Alarms[45]
          TriggerValues:
            [0] = 1
    [60]:
      Name = Alarm46
      Message = {$Alarms/Alarm.46}
      Code = 46
      Behavior = DiscreteValueMonitoring
        Monitoring:
          MonitoredPV = ::AlarmMgt:Alarms[46]
          TriggerValues:
            [0] = 1
    [61]:
      Name = Alarm47
      Message = {$Alarms/Alarm.47}
      Code = 47
      Behavior = DiscreteValueMonitoring
        Monitoring:
          MonitoredPV = ::AlarmMgt:Alarms[47]
          TriggerValues:
            [0] = 1
    [62]:
      Name = Alarm48
      Message = {$Alarms/Alarm.48}
      Code = 48
      Behavior = DiscreteValueMonitoring
        Monitoring:
          MonitoredPV = ::AlarmMgt:Alarms[48]
          TriggerValues:
            [0] = 1
    [63]:
      Name = Alarm49
      Message = {$Alarms/Alarm.49}
      Code = 49
      Behavior = DiscreteValueMonitoring
        Monitoring:
          MonitoredPV = ::AlarmMgt:Alarms[49]
          TriggerValues:
            [0] = 1
    [64]:
      Name = Alarm50
      Message = {$Alarms/Alarm.50}
      Behavior = DiscreteValueMonitoring
        Monitoring:
          MonitoredPV = ::AlarmMgt:Alarms[50]
          TriggerValues:
            [0] = 1
    [65]:
      Name = Alarm51
      Message = {$Alarms/Alarm.51}
      Code = 51
      Behavior = DiscreteValueMonitoring
        Monitoring:
          MonitoredPV = ::AlarmMgt:Alarms[51]
          TriggerValues:
            [0] = 1
    [66]:
      Name = Alarm52
      Message = {$Alarms/Alarm.52}
      Code = 52
      Behavior = DiscreteValueMonitoring
        Monitoring:
          MonitoredPV = ::AlarmMgt:Alarms[52]
          TriggerValues:
            [0] = 1
    [67]:
      Name = Alarm53
      Message = {$Alarms/Alarm.53}
      Code = 53
      Behavior = DiscreteValueMonitoring
        Monitoring:
          MonitoredPV = ::AlarmMgt:Alarms[53]
          TriggerValues:
            [0] = 1
    [68]:
      Name = Alarm54
      Message = {$Alarms/Alarm.54}
      Code = 54
      Behavior = DiscreteValueMonitoring
        Monitoring:
          MonitoredPV = ::AlarmMgt:Alarms[54]
          TriggerValues:
            [0] = 1
    [69]:
      Name = Alarm55
      Message = {$Alarms/Alarm.55}
      Code = 55
      Behavior = DiscreteValueMonitoring
        Monitoring:
          MonitoredPV = ::AlarmMgt:Alarms[55]
          TriggerValues:
            [0] = 1
    [70]:
      Name = Alarm56
      Message = {$Alarms/Alarm.56}
      Code = 56
      Behavior = DiscreteValueMonitoring
        Monitoring:
          MonitoredPV = ::AlarmMgt:Alarms[56]
          TriggerValues:
            [0] = 1
    [71]:
      Name = Alarm57
      Message = {$Alarms/Alarm.57}
      Code = 57
      Behavior = DiscreteValueMonitoring
        Monitoring:
          MonitoredPV = ::AlarmMgt:Alarms[57]
          TriggerValues:
            [0] = 1
    [72]:
      Name = Alarm58
      Message = {$Alarms/Alarm.58}
      Code = 58
      Behavior = DiscreteValueMonitoring
        Monitoring:
          MonitoredPV = ::AlarmMgt:Alarms[58]
          TriggerValues:
            [0] = 1
    [73]:
      Name = Alarm59
      Message = {$Alarms/Alarm.59}
      Code = 59
      Behavior = DiscreteValueMonitoring
        Monitoring:
          MonitoredPV = ::AlarmMgt:Alarms[59]
          TriggerValues:
            [0] = 1
    [74]:
      Name = Alarm60
      Message = {$Alarms/Alarm.60}
      Behavior = DiscreteValueMonitoring
        Monitoring:
          MonitoredPV = ::AlarmMgt:Alarms[60]
          TriggerValues:
            [0] = 1
    [75]:
      Name = Alarm61
      Message = {$Alarms/Alarm.61}
      Code = 61
      Behavior = DiscreteValueMonitoring
        Monitoring:
          MonitoredPV = ::AlarmMgt:Alarms[61]
          TriggerValues:
            [0] = 1
    [76]:
      Name = Alarm62
      Message = {$Alarms/Alarm.62}
      Code = 62
      Behavior = DiscreteValueMonitoring
        Monitoring:
          MonitoredPV = ::AlarmMgt:Alarms[62]
          TriggerValues:
            [0] = 1
    [77]:
      Name = Alarm63
      Message = {$Alarms/Alarm.63}
      Code = 63
      Behavior = DiscreteValueMonitoring
        Monitoring:
          MonitoredPV = ::AlarmMgt:Alarms[63]
          TriggerValues:
            [0] = 1
    [78]:
      Name = Alarm64
      Message = {$Alarms/Alarm.64}
      Code = 64
      Behavior = DiscreteValueMonitoring
        Monitoring:
          MonitoredPV = ::AlarmMgt:Alarms[64]
          TriggerValues:
            [0] = 1
    [79]:
      Name = Alarm65
      Message = {$Alarms/Alarm.65}
      Code = 65
      Behavior = DiscreteValueMonitoring
        Monitoring:
          MonitoredPV = ::AlarmMgt:Alarms[65]
          TriggerValues:
            [0] = 1
    [80]:
      Name = Alarm66
      Message = {$Alarms/Alarm.66}
      Code = 66
      Behavior = DiscreteValueMonitoring
        Monitoring:
          MonitoredPV = ::AlarmMgt:Alarms[66]
          TriggerValues:
            [0] = 1
    [81]:
      Name = Alarm67
      Message = {$Alarms/Alarm.67}
      Code = 67
      Behavior = DiscreteValueMonitoring
        Monitoring:
          MonitoredPV = ::AlarmMgt:Alarms[67]
          TriggerValues:
            [0] = 1
    [82]:
      Name = Alarm68
      Message = {$Alarms/Alarm.68}
      Code = 68
      Behavior = DiscreteValueMonitoring
        Monitoring:
          MonitoredPV = ::AlarmMgt:Alarms[68]
          TriggerValues:
            [0] = 1
    [83]:
      Name = Alarm69
      Message = {$Alarms/Alarm.69}
      Code = 69
      Behavior = DiscreteValueMonitoring
        Monitoring:
          MonitoredPV = ::AlarmMgt:Alarms[69]
          TriggerValues:
            [0] = 1
    [84]:
      Name = Alarm70
      Message = {$Alarms/Alarm.70}
      Behavior = DiscreteValueMonitoring
        Monitoring:
          MonitoredPV = ::AlarmMgt:Alarms[70]
          TriggerValues:
            [0] = 1
    [85]:
      Name = Alarm71
      Message = {$Alarms/Alarm.71}
      Code = 71
      Behavior = DiscreteValueMonitoring
        Monitoring:
          MonitoredPV = ::AlarmMgt:Alarms[71]
          TriggerValues:
            [0] = 1
    [86]:
      Name = Alarm72
      Message = {$Alarms/Alarm.72}
      Code = 72
      Behavior = DiscreteValueMonitoring
        Monitoring:
          MonitoredPV = ::AlarmMgt:Alarms[72]
          TriggerValues:
            [0] = 1
    [87]:
      Name = Alarm73
      Message = {$Alarms/Alarm.73}
      Code = 73
      Behavior = DiscreteValueMonitoring
        Monitoring:
          MonitoredPV = ::AlarmMgt:Alarms[73]
          TriggerValues:
            [0] = 1
    [88]:
      Name = Alarm74
      Message = {$Alarms/Alarm.74}
      Code = 74
      Behavior = DiscreteValueMonitoring
        Monitoring:
          MonitoredPV = ::AlarmMgt:Alarms[74]
          TriggerValues:
            [0] = 1
    [89]:
      Name = Alarm75
      Message = {$Alarms/Alarm.75}
      Code = 75
      Behavior = DiscreteValueMonitoring
        Monitoring:
          MonitoredPV = ::AlarmMgt:Alarms[75]
          TriggerValues:
            [0] = 1
    [90]:
      Name = Alarm76
      Message = {$Alarms/Alarm.76}
      Code = 76
      Behavior = DiscreteValueMonitoring
        Monitoring:
          MonitoredPV = ::AlarmMgt:Alarms[76]
          TriggerValues:
            [0] = 1
    [91]:
      Name = Alarm77
      Message = {$Alarms/Alarm.77}
      Code = 77
      Behavior = DiscreteValueMonitoring
        Monitoring:
          MonitoredPV = ::AlarmMgt:Alarms[77]
          TriggerValues:
            [0] = 1
    [92]:
      Name = Alarm78
      Message = {$Alarms/Alarm.78}
      Code = 78
      Behavior = DiscreteValueMonitoring
        Monitoring:
          MonitoredPV = ::AlarmMgt:Alarms[78]
          TriggerValues:
            [0] = 1
    [93]:
      Name = Alarm79
      Message = {$Alarms/Alarm.79}
      Code = 79
      Behavior = DiscreteValueMonitoring
        Monitoring:
          MonitoredPV = ::AlarmMgt:Alarms[79]
          TriggerValues:
            [0] = 1
    [94]:
      Name = Alarm80
      Message = {$Alarms/Alarm.80}
      Behavior = DiscreteValueMonitoring
        Monitoring:
          MonitoredPV = ::AlarmMgt:Alarms[80]
          TriggerValues:
            [0] = 1
    [95]:
      Name = Alarm81
      Message = {$Alarms/Alarm.81}
      Code = 81
      Behavior = DiscreteValueMonitoring
        Monitoring:
          MonitoredPV = ::AlarmMgt:Alarms[81]
          TriggerValues:
            [0] = 1
    [96]:
      Name = Alarm82
      Message = {$Alarms/Alarm.82}
      Code = 82
      Behavior = DiscreteValueMonitoring
        Monitoring:
          MonitoredPV = ::AlarmMgt:Alarms[82]
          TriggerValues:
            [0] = 1
    [97]:
      Name = Alarm83
      Message = {$Alarms/Alarm.83}
      Code = 83
      Behavior = DiscreteValueMonitoring
        Monitoring:
          MonitoredPV = ::AlarmMgt:Alarms[83]
          TriggerValues:
            [0] = 1
    [98]:
      Name = Alarm84
      Message = {$Alarms/Alarm.84}
      Code = 84
      Behavior = DiscreteValueMonitoring
        Monitoring:
          MonitoredPV = ::AlarmMgt:Alarms[84]
          TriggerValues:
            [0] = 1
    [99]:
      Name = Alarm85
      Message = {$Alarms/Alarm.85}
      Code = 85
      Behavior = DiscreteValueMonitoring
        Monitoring:
          MonitoredPV = ::AlarmMgt:Alarms[85]
          TriggerValues:
            [0] = 1
    [100]:
      Name = Alarm86
      Message = {$Alarms/Alarm.86}
      Code = 86
      Behavior = DiscreteValueMonitoring
        Monitoring:
          MonitoredPV = ::AlarmMgt:Alarms[86]
          TriggerValues:
            [0] = 1
    [101]:
      Name = Alarm87
      Message = {$Alarms/Alarm.87}
      Code = 87
      Behavior = DiscreteValueMonitoring
        Monitoring:
          MonitoredPV = ::AlarmMgt:Alarms[87]
          TriggerValues:
            [0] = 1
    [102]:
      Name = Alarm88
      Message = {$Alarms/Alarm.88}
      Code = 88
      Behavior = DiscreteValueMonitoring
        Monitoring:
          MonitoredPV = ::AlarmMgt:Alarms[88]
          TriggerValues:
            [0] = 1
    [103]:
      Name = Alarm89
      Message = {$Alarms/Alarm.89}
      Code = 89
      Behavior = DiscreteValueMonitoring
        Monitoring:
          MonitoredPV = ::AlarmMgt:Alarms[89]
          TriggerValues:
            [0] = 1
    [104]:
      Name = Alarm90
      Message = {$Alarms/Alarm.90}
      Behavior = DiscreteValueMonitoring
        Monitoring:
          MonitoredPV = ::AlarmMgt:Alarms[90]
          TriggerValues:
            [0] = 1
    [105]:
      Name = Alarm91
      Message = {$Alarms/Alarm.91}
      Code = 91
      Behavior = DiscreteValueMonitoring
        Monitoring:
          MonitoredPV = ::AlarmMgt:Alarms[91]
          TriggerValues:
            [0] = 1
    [106]:
      Name = Alarm92
      Message = {$Alarms/Alarm.92}
      Code = 92
      Behavior = DiscreteValueMonitoring
        Monitoring:
          MonitoredPV = ::AlarmMgt:Alarms[92]
          TriggerValues:
            [0] = 1
    [107]:
      Name = Alarm93
      Message = {$Alarms/Alarm.93}
      Code = 93
      Behavior = DiscreteValueMonitoring
        Monitoring:
          MonitoredPV = ::AlarmMgt:Alarms[93]
          TriggerValues:
            [0] = 1
    [108]:
      Name = Alarm94
      Message = {$Alarms/Alarm.94}
      Code = 94
      Behavior = DiscreteValueMonitoring
        Monitoring:
          MonitoredPV = ::AlarmMgt:Alarms[94]
          TriggerValues:
            [0] = 1
    [109]:
      Name = Alarm95
      Message = {$Alarms/Alarm.95}
      Code = 95
      Behavior = DiscreteValueMonitoring
        Monitoring:
          MonitoredPV = ::AlarmMgt:Alarms[95]
          TriggerValues:
            [0] = 1
    [110]:
      Name = Alarm96
      Message = {$Alarms/Alarm.96}
      Code = 96
      Behavior = DiscreteValueMonitoring
        Monitoring:
          MonitoredPV = ::AlarmMgt:Alarms[96]
          TriggerValues:
            [0] = 1
    [111]:
      Name = Alarm97
      Message = {$Alarms/Alarm.97}
      Code = 97
      Behavior = DiscreteValueMonitoring
        Monitoring:
          MonitoredPV = ::AlarmMgt:Alarms[97]
          TriggerValues:
            [0] = 1
    [112]:
      Name = Alarm98
      Message = {$Alarms/Alarm.98}
      Code = 98
      Behavior = DiscreteValueMonitoring
        Monitoring:
          MonitoredPV = ::AlarmMgt:Alarms[98]
          TriggerValues:
            [0] = 1
    [113]:
      Name = Alarm99
      Message = {$Alarms/Alarm.99}
      Code = 99
      Behavior = DiscreteValueMonitoring
        Monitoring:
          MonitoredPV = ::AlarmMgt:Alarms[99]
          TriggerValues:
            [0] = 1
  mapp.AlarmX.Core.Snippets:
    AutoDetect = 1
    [0]:
      Key = snippet1
      Value:
        PV = ::AlarmMgt:AlarmExamples.SnippetValue
  mapp.AlarmX.Core.Queries:
    [0]:
      Name = ActiveAlarms
      Update = ::AlarmMgt:AlarmQuery.ActiveAlarmUpdateCount
      Source:
        SELECT:
          [0]:
            PV = ::AlarmMgt:AlarmQuery.Alarms[].Name
          [1]:
            Column = Message
            PV = ::AlarmMgt:AlarmQuery.Alarms[].Message
          [2]:
            Column = Code
            PV = ::AlarmMgt:AlarmQuery.Alarms[].Code
          [3]:
            Column = Severity
            PV = ::AlarmMgt:AlarmQuery.Alarms[].Severity
          [4]:
            Column = Scope
            PV = ::AlarmMgt:AlarmQuery.Alarms[].Scope
          [5]:
            Column = TimeStamp
            PV = ::AlarmMgt:AlarmQuery.Alarms[].TimeStamp
          [6]:
            Column = AdditionalInformation1
            PV = ::AlarmMgt:AlarmQuery.Alarms[].AdditionalInfo
          [7]:
            Column = StateActive
            PV = ::AlarmMgt:AlarmQuery.Alarms[].Active
          [8]:
            Column = StateAcknowledged
            PV = ::AlarmMgt:AlarmQuery.Alarms[].Acknowledged
```

### AlarmXCfg.mpalarmxcore - 5PPC2200_AL14_000/mappServices/AlarmX/AlarmXCfg.mpalarmxcore
```
Element gMpLinkAlarmXCore (Type=mpalarmxcore)
  mapp.AlarmX.Core:
    BySeverity:
      [0]:
        Severity = 1..9
        [0] = Reaction
          Name = Info
      [1]:
        Severity = 10..19
        [0] = Reaction
          Name = Warning
      [2]:
        Severity = 20..29
        [0] = Reaction
          Name = Error
  mapp.AlarmX.Core.Configuration:
    [0]:
      Name = EmergencyStop_0
      Message = {$Alarms/EmergencyStop.0}
      Severity = 29
      Behavior = DiscreteValueMonitoring
        Monitoring:
          MonitoredPV = ::AlarmMgr:SafetyInputs.EmergencyStop[0]
          TriggerValues:
            [0] = 1
    [1]:
      Name = EmergencyStop_1
      Message = {$Alarms/EmergencyStop.1}
      Behavior = DiscreteValueMonitoring
        Monitoring:
          MonitoredPV = ::AlarmMgr:SafetyInputs.EmergencyStop[1]
          TriggerValues:
            [0] = 1
    [2]:
      Name = EmergencyStop_2
      Message = {$Alarms/EmergencyStop.2}
      Behavior = DiscreteValueMonitoring
        Monitoring:
          MonitoredPV = ::AlarmMgr:SafetyInputs.EmergencyStop[2]
          TriggerValues:
            [0] = 1
    [3]:
      Name = SafetyDoor_0
      Message = {$Alarms/SafetyDoor.0}
      Severity = 29
      Behavior = DiscreteValueMonitoring
        Monitoring:
          MonitoredPV = ::AlarmMgr:SafetyInputs.SafetyDoor[0]
          TriggerValues:
            [0] = 1
    [4]:
      Name = SafetyDoor_1
      Message = {$Alarms/SafetyDoor.1}
      Severity = 29
      Behavior = DiscreteValueMonitoring
        Monitoring:
          MonitoredPV = ::AlarmMgr:SafetyInputs.SafetyDoor[1]
          TriggerValues:
            [0] = 1
    [5]:
      Name = SafetyDoor_2
      Message = {$Alarms/SafetyDoor.2}
      Severity = 29
      Behavior = DiscreteValueMonitoring
        Monitoring:
          MonitoredPV = ::AlarmMgr:SafetyInputs.SafetyDoor[2]
          TriggerValues:
            [0] = 1
    [6]:
      Name = SafetyDoor_3
      Message = {$Alarms/SafetyDoor.3}
      Severity = 29
      Behavior = DiscreteValueMonitoring
        Monitoring:
          MonitoredPV = ::AlarmMgr:SafetyInputs.SafetyDoor[3]
          TriggerValues:
            [0] = 1
    [7]:
      Name = SafetyDoor_4
      Message = {$Alarms/SafetyDoor.4}
      Severity = 29
      Behavior = DiscreteValueMonitoring
        Monitoring:
          MonitoredPV = ::AlarmMgr:SafetyInputs.SafetyDoor[4]
          TriggerValues:
            [0] = 1
    [8]:
      Name = SafetyDoor_5
      Message = {$Alarms/SafetyDoor.5}
      Severity = 29
      Behavior = DiscreteValueMonitoring
        Monitoring:
          MonitoredPV = ::AlarmMgr:SafetyInputs.SafetyDoor[5]
          TriggerValues:
            [0] = 1
    [9]:
      Name = LevelMonitoringExample
      Message = {$Alarms/LevelMonitoringAlarmExample} {=$Alarms/{&LimitText}}
      Behavior = LevelMonitoring
        Monitoring:
          MonitoredPV = ::AlarmMgr:AlarmExamples.LevelMonitoring
          LowLimitEnable = Static
            Limit = 20
            LimitText = LevelMonitoringAlarmLowTextExample
            LowLowLimitEnable = Static
              Limit = 10
              LimitText = LevelMonitoringAlarmLowLowTextExample
          HighLimitEnable = Static
            Limit = 80
            LimitText = LevelMonitoringAlarmHighTextExample
            HighHighLimitEnable = Static
              Limit = 90
              LimitText = LevelMonitoringAlarmHighHighTextExample
    [10]:
      Name = DeviationMonitoringExample
      Message = {$Alarms/DeviationMonitoringAlarmExample} {&LimitText}
      Behavior = DeviationMonitoring
        Monitoring:
          MonitoredPV = ::AlarmMgr:AlarmExamples.DeviationMonitoring
          SetpointPV = ::AlarmMgr:AlarmExamples.DeviationMonitoringSetpoint
          LowLimitEnable = Static
            Limit = -5
            LimitText = Low limit exceeded
          HighLimitEnable = Static
            Limit = 5
            LimitText = High limit exceeded
    [11]:
      Name = RateOfChangeExample
      Message = {$Alarms/RateOfChangeAlarmExample}
      Behavior = RateOfChangeMonitoring
        Monitoring:
          MonitoredPV = ::AlarmMgr:AlarmExamples.RateOfChange
          HighLimitEnable = Static
            Limit = 5
            LimitText = High limit exceeded
    [12]:
      Name = SnippetExample
      Message = Show a snippet directly: {&snippet1}. Show from localizable text: {$Alarms/SnippetExample}
      Behavior = DiscreteValueMonitoring
        Monitoring:
          MonitoredPV = ::AlarmMgr:AlarmExamples.SnippetValue
          TriggerValues:
            [0] = 50..100
    [13]:
      Name = MpAlarmXControlExample
      Message = {$Alarms/MpAlarmXControlExample}
      Severity = 20
      Behavior:
        Async = TRUE
    [14]:
      Name = Alarm0
      Message = {$Alarms/Alarm.0}
      Behavior = DiscreteValueMonitoring
        Monitoring:
          MonitoredPV = ::AlarmMgr:Alarms[0]
          InhibitPV = ::AlarmMgr:CommissioningModeActive
          TriggerValues:
            [0] = 1
    [15]:
      Name = Alarm1
      Message = {$Alarms/Alarm.1}
      Code = 1
      Behavior = DiscreteValueMonitoring
        Monitoring:
          MonitoredPV = ::AlarmMgr:Alarms[1]
          TriggerValues:
            [0] = 1
    [16]:
      Name = Alarm2
      Message = {$Alarms/Alarm.2}
      Code = 2
      Behavior = DiscreteValueMonitoring
        Monitoring:
          MonitoredPV = ::AlarmMgr:Alarms[2]
          TriggerValues:
            [0] = 1
    [17]:
      Name = Alarm3
      Message = {$Alarms/Alarm.3}
      Code = 3
      Behavior = DiscreteValueMonitoring
        Monitoring:
          MonitoredPV = ::AlarmMgr:Alarms[3]
          TriggerValues:
            [0] = 1
    [18]:
      Name = Alarm4
      Message = {$Alarms/Alarm.4}
      Code = 4
      Behavior = DiscreteValueMonitoring
        Monitoring:
          MonitoredPV = ::AlarmMgr:Alarms[4]
          TriggerValues:
            [0] = 1
    [19]:
      Name = Alarm5
      Message = {$Alarms/Alarm.5}
      Code = 5
      Behavior = DiscreteValueMonitoring
        Monitoring:
          MonitoredPV = ::AlarmMgr:Alarms[5]
          TriggerValues:
            [0] = 1
    [20]:
      Name = Alarm6
      Message = {$Alarms/Alarm.6}
      Code = 6
      Behavior = DiscreteValueMonitoring
        Monitoring:
          MonitoredPV = ::AlarmMgr:Alarms[6]
          TriggerValues:
            [0] = 1
    [21]:
      Name = Alarm7
      Message = {$Alarms/Alarm.7}
      Code = 7
      Behavior = DiscreteValueMonitoring
        Monitoring:
          MonitoredPV = ::AlarmMgr:Alarms[7]
          TriggerValues:
            [0] = 1
    [22]:
      Name = Alarm8
      Message = {$Alarms/Alarm.8}
      Code = 8
      Behavior = DiscreteValueMonitoring
        Monitoring:
          MonitoredPV = ::AlarmMgr:Alarms[8]
          TriggerValues:
            [0] = 1
    [23]:
      Name = Alarm9
      Message = {$Alarms/Alarm.9}
      Code = 9
      Behavior = DiscreteValueMonitoring
        Monitoring:
          MonitoredPV = ::AlarmMgr:Alarms[9]
          TriggerValues:
            [0] = 1
    [24]:
      Name = Alarm10
      Message = {$Alarms/Alarm.10}
      Code = 10
      Behavior = DiscreteValueMonitoring
        Monitoring:
          MonitoredPV = ::AlarmMgr:Alarms[10]
          TriggerValues:
            [0] = 1
    [25]:
      Name = Alarm11
      Message = {$Alarms/Alarm.11}
      Code = 11
      Behavior = DiscreteValueMonitoring
        Monitoring:
          MonitoredPV = ::AlarmMgr:Alarms[11]
          TriggerValues:
            [0] = 1
    [26]:
      Name = Alarm12
      Message = {$Alarms/Alarm.12}
      Code = 12
      Behavior = DiscreteValueMonitoring
        Monitoring:
          MonitoredPV = ::AlarmMgr:Alarms[12]
          TriggerValues:
            [0] = 1
    [27]:
      Name = Alarm13
      Message = {$Alarms/Alarm.13}
      Code = 13
      Behavior = DiscreteValueMonitoring
        Monitoring:
          MonitoredPV = ::AlarmMgr:Alarms[13]
          TriggerValues:
            [0] = 1
    [28]:
      Name = Alarm14
      Message = {$Alarms/Alarm.14}
      Code = 14
      Behavior = DiscreteValueMonitoring
        Monitoring:
          MonitoredPV = ::AlarmMgr:Alarms[14]
          TriggerValues:
            [0] = 1
    [29]:
      Name = Alarm15
      Message = {$Alarms/Alarm.15}
      Code = 15
      Behavior = DiscreteValueMonitoring
        Monitoring:
          MonitoredPV = ::AlarmMgr:Alarms[15]
          TriggerValues:
            [0] = 1
    [30]:
      Name = Alarm16
      Message = {$Alarms/Alarm.16}
      Code = 16
      Behavior = DiscreteValueMonitoring
        Monitoring:
          MonitoredPV = ::AlarmMgr:Alarms[16]
          TriggerValues:
            [0] = 1
    [31]:
      Name = Alarm17
      Message = {$Alarms/Alarm.17}
      Code = 17
      Behavior = DiscreteValueMonitoring
        Monitoring:
          MonitoredPV = ::AlarmMgr:Alarms[17]
          TriggerValues:
            [0] = 1
    [32]:
      Name = Alarm18
      Message = {$Alarms/Alarm.18}
      Code = 18
      Behavior = DiscreteValueMonitoring
        Monitoring:
          MonitoredPV = ::AlarmMgr:Alarms[18]
          TriggerValues:
            [0] = 1
    [33]:
      Name = Alarm19
      Message = {$Alarms/Alarm.19}
      Code = 19
      Behavior = DiscreteValueMonitoring
        Monitoring:
          MonitoredPV = ::AlarmMgr:Alarms[19]
          TriggerValues:
            [0] = 1
    [34]:
      Name = Alarm20
      Message = {$Alarms/Alarm.20}
      Behavior = DiscreteValueMonitoring
        Monitoring:
          MonitoredPV = ::AlarmMgr:Alarms[20]
          TriggerValues:
            [0] = 1
    [35]:
      Name = Alarm21
      Message = {$Alarms/Alarm.21}
      Code = 21
      Behavior = DiscreteValueMonitoring
        Monitoring:
          MonitoredPV = ::AlarmMgr:Alarms[21]
          TriggerValues:
            [0] = 1
    [36]:
      Name = Alarm22
      Message = {$Alarms/Alarm.22}
      Code = 22
      Behavior = DiscreteValueMonitoring
        Monitoring:
          MonitoredPV = ::AlarmMgr:Alarms[22]
          TriggerValues:
            [0] = 1
    [37]:
      Name = Alarm23
      Message = {$Alarms/Alarm.23}
      Code = 23
      Behavior = DiscreteValueMonitoring
        Monitoring:
          MonitoredPV = ::AlarmMgr:Alarms[23]
          TriggerValues:
            [0] = 1
    [38]:
      Name = Alarm24
      Message = {$Alarms/Alarm.24}
      Code = 24
      Behavior = DiscreteValueMonitoring
        Monitoring:
          MonitoredPV = ::AlarmMgr:Alarms[24]
          TriggerValues:
            [0] = 1
    [39]:
      Name = Alarm25
      Message = {$Alarms/Alarm.25}
      Code = 25
      Behavior = DiscreteValueMonitoring
        Monitoring:
          MonitoredPV = ::AlarmMgr:Alarms[25]
          TriggerValues:
            [0] = 1
    [40]:
      Name = Alarm26
      Message = {$Alarms/Alarm.26}
      Code = 26
      Behavior = DiscreteValueMonitoring
        Monitoring:
          MonitoredPV = ::AlarmMgr:Alarms[26]
          TriggerValues:
            [0] = 1
    [41]:
      Name = Alarm27
      Message = {$Alarms/Alarm.27}
      Code = 27
      Behavior = DiscreteValueMonitoring
        Monitoring:
          MonitoredPV = ::AlarmMgr:Alarms[27]
          TriggerValues:
            [0] = 1
    [42]:
      Name = Alarm28
      Message = {$Alarms/Alarm.28}
      Code = 28
      Behavior = DiscreteValueMonitoring
        Monitoring:
          MonitoredPV = ::AlarmMgr:Alarms[28]
          TriggerValues:
            [0] = 1
    [43]:
      Name = Alarm29
      Message = {$Alarms/Alarm.29}
      Code = 29
      Behavior = DiscreteValueMonitoring
        Monitoring:
          MonitoredPV = ::AlarmMgr:Alarms[29]
          TriggerValues:
            [0] = 1
    [44]:
      Name = Alarm30
      Message = {$Alarms/Alarm.30}
      Behavior = DiscreteValueMonitoring
        Monitoring:
          MonitoredPV = ::AlarmMgr:Alarms[30]
          TriggerValues:
            [0] = 1
    [45]:
      Name = Alarm31
      Message = {$Alarms/Alarm.31}
      Code = 31
      Behavior = DiscreteValueMonitoring
        Monitoring:
          MonitoredPV = ::AlarmMgr:Alarms[31]
          TriggerValues:
            [0] = 1
    [46]:
      Name = Alarm32
      Message = {$Alarms/Alarm.32}
      Code = 32
      Behavior = DiscreteValueMonitoring
        Monitoring:
          MonitoredPV = ::AlarmMgr:Alarms[32]
          TriggerValues:
            [0] = 1
    [47]:
      Name = Alarm33
      Message = {$Alarms/Alarm.33}
      Code = 33
      Behavior = DiscreteValueMonitoring
        Monitoring:
          MonitoredPV = ::AlarmMgr:Alarms[33]
          TriggerValues:
            [0] = 1
    [48]:
      Name = Alarm34
      Message = {$Alarms/Alarm.34}
      Code = 34
      Behavior = DiscreteValueMonitoring
        Monitoring:
          MonitoredPV = ::AlarmMgr:Alarms[34]
          TriggerValues:
            [0] = 1
    [49]:
      Name = Alarm35
      Message = {$Alarms/Alarm.35}
      Code = 35
      Behavior = DiscreteValueMonitoring
        Monitoring:
          MonitoredPV = ::AlarmMgr:Alarms[35]
          TriggerValues:
            [0] = 1
    [50]:
      Name = Alarm36
      Message = {$Alarms/Alarm.36}
      Code = 36
      Behavior = DiscreteValueMonitoring
        Monitoring:
          MonitoredPV = ::AlarmMgr:Alarms[36]
          TriggerValues:
            [0] = 1
    [51]:
      Name = Alarm37
      Message = {$Alarms/Alarm.37}
      Code = 37
      Behavior = DiscreteValueMonitoring
        Monitoring:
          MonitoredPV = ::AlarmMgr:Alarms[37]
          TriggerValues:
            [0] = 1
    [52]:
      Name = Alarm38
      Message = {$Alarms/Alarm.38}
      Code = 38
      Behavior = DiscreteValueMonitoring
        Monitoring:
          MonitoredPV = ::AlarmMgr:Alarms[38]
          TriggerValues:
            [0] = 1
    [53]:
      Name = Alarm39
      Message = {$Alarms/Alarm.39}
      Code = 39
      Behavior = DiscreteValueMonitoring
        Monitoring:
          MonitoredPV = ::AlarmMgr:Alarms[39]
          TriggerValues:
            [0] = 1
    [54]:
      Name = Alarm40
      Message = {$Alarms/Alarm.40}
      Behavior = DiscreteValueMonitoring
        Monitoring:
          MonitoredPV = ::AlarmMgr:Alarms[40]
          TriggerValues:
            [0] = 1
    [55]:
      Name = Alarm41
      Message = {$Alarms/Alarm.41}
      Code = 41
      Behavior = DiscreteValueMonitoring
        Monitoring:
          MonitoredPV = ::AlarmMgr:Alarms[41]
          TriggerValues:
            [0] = 1
    [56]:
      Name = Alarm42
      Message = {$Alarms/Alarm.42}
      Code = 42
      Behavior = DiscreteValueMonitoring
        Monitoring:
          MonitoredPV = ::AlarmMgr:Alarms[42]
          TriggerValues:
            [0] = 1
    [57]:
      Name = Alarm43
      Message = {$Alarms/Alarm.43}
      Code = 43
      Behavior = DiscreteValueMonitoring
        Monitoring:
          MonitoredPV = ::AlarmMgr:Alarms[43]
          TriggerValues:
            [0] = 1
    [58]:
      Name = Alarm44
      Message = {$Alarms/Alarm.44}
      Code = 44
      Behavior = DiscreteValueMonitoring
        Monitoring:
          MonitoredPV = ::AlarmMgr:Alarms[44]
          TriggerValues:
            [0] = 1
    [59]:
      Name = Alarm45
      Message = {$Alarms/Alarm.45}
      Code = 45
      Behavior = DiscreteValueMonitoring
        Monitoring:
          MonitoredPV = ::AlarmMgr:Alarms[45]
          TriggerValues:
            [0] = 1
    [60]:
      Name = Alarm46
      Message = {$Alarms/Alarm.46}
      Code = 46
      Behavior = DiscreteValueMonitoring
        Monitoring:
          MonitoredPV = ::AlarmMgr:Alarms[46]
          TriggerValues:
            [0] = 1
    [61]:
      Name = Alarm47
      Message = {$Alarms/Alarm.47}
      Code = 47
      Behavior = DiscreteValueMonitoring
        Monitoring:
          MonitoredPV = ::AlarmMgr:Alarms[47]
          TriggerValues:
            [0] = 1
    [62]:
      Name = Alarm48
      Message = {$Alarms/Alarm.48}
      Code = 48
      Behavior = DiscreteValueMonitoring
        Monitoring:
          MonitoredPV = ::AlarmMgr:Alarms[48]
          TriggerValues:
            [0] = 1
    [63]:
      Name = Alarm49
      Message = {$Alarms/Alarm.49}
      Code = 49
      Behavior = DiscreteValueMonitoring
        Monitoring:
          MonitoredPV = ::AlarmMgr:Alarms[49]
          TriggerValues:
            [0] = 1
    [64]:
      Name = Alarm50
      Message = {$Alarms/Alarm.50}
      Behavior = DiscreteValueMonitoring
        Monitoring:
          MonitoredPV = ::AlarmMgr:Alarms[50]
          TriggerValues:
            [0] = 1
    [65]:
      Name = Alarm51
      Message = {$Alarms/Alarm.51}
      Code = 51
      Behavior = DiscreteValueMonitoring
        Monitoring:
          MonitoredPV = ::AlarmMgr:Alarms[51]
          TriggerValues:
            [0] = 1
    [66]:
      Name = Alarm52
      Message = {$Alarms/Alarm.52}
      Code = 52
      Behavior = DiscreteValueMonitoring
        Monitoring:
          MonitoredPV = ::AlarmMgr:Alarms[52]
          TriggerValues:
            [0] = 1
    [67]:
      Name = Alarm53
      Message = {$Alarms/Alarm.53}
      Code = 53
      Behavior = DiscreteValueMonitoring
        Monitoring:
          MonitoredPV = ::AlarmMgr:Alarms[53]
          TriggerValues:
            [0] = 1
    [68]:
      Name = Alarm54
      Message = {$Alarms/Alarm.54}
      Code = 54
      Behavior = DiscreteValueMonitoring
        Monitoring:
          MonitoredPV = ::AlarmMgr:Alarms[54]
          TriggerValues:
            [0] = 1
    [69]:
      Name = Alarm55
      Message = {$Alarms/Alarm.55}
      Code = 55
      Behavior = DiscreteValueMonitoring
        Monitoring:
          MonitoredPV = ::AlarmMgr:Alarms[55]
          TriggerValues:
            [0] = 1
    [70]:
      Name = Alarm56
      Message = {$Alarms/Alarm.56}
      Code = 56
      Behavior = DiscreteValueMonitoring
        Monitoring:
          MonitoredPV = ::AlarmMgr:Alarms[56]
          TriggerValues:
            [0] = 1
    [71]:
      Name = Alarm57
      Message = {$Alarms/Alarm.57}
      Code = 57
      Behavior = DiscreteValueMonitoring
        Monitoring:
          MonitoredPV = ::AlarmMgr:Alarms[57]
          TriggerValues:
            [0] = 1
    [72]:
      Name = Alarm58
      Message = {$Alarms/Alarm.58}
      Code = 58
      Behavior = DiscreteValueMonitoring
        Monitoring:
          MonitoredPV = ::AlarmMgr:Alarms[58]
          TriggerValues:
            [0] = 1
    [73]:
      Name = Alarm59
      Message = {$Alarms/Alarm.59}
      Code = 59
      Behavior = DiscreteValueMonitoring
        Monitoring:
          MonitoredPV = ::AlarmMgr:Alarms[59]
          TriggerValues:
            [0] = 1
    [74]:
      Name = Alarm60
      Message = {$Alarms/Alarm.60}
      Behavior = DiscreteValueMonitoring
        Monitoring:
          MonitoredPV = ::AlarmMgr:Alarms[60]
          TriggerValues:
            [0] = 1
    [75]:
      Name = Alarm61
      Message = {$Alarms/Alarm.61}
      Code = 61
      Behavior = DiscreteValueMonitoring
        Monitoring:
          MonitoredPV = ::AlarmMgr:Alarms[61]
          TriggerValues:
            [0] = 1
    [76]:
      Name = Alarm62
      Message = {$Alarms/Alarm.62}
      Code = 62
      Behavior = DiscreteValueMonitoring
        Monitoring:
          MonitoredPV = ::AlarmMgr:Alarms[62]
          TriggerValues:
            [0] = 1
    [77]:
      Name = Alarm63
      Message = {$Alarms/Alarm.63}
      Code = 63
      Behavior = DiscreteValueMonitoring
        Monitoring:
          MonitoredPV = ::AlarmMgr:Alarms[63]
          TriggerValues:
            [0] = 1
    [78]:
      Name = Alarm64
      Message = {$Alarms/Alarm.64}
      Code = 64
      Behavior = DiscreteValueMonitoring
        Monitoring:
          MonitoredPV = ::AlarmMgr:Alarms[64]
          TriggerValues:
            [0] = 1
    [79]:
      Name = Alarm65
      Message = {$Alarms/Alarm.65}
      Code = 65
      Behavior = DiscreteValueMonitoring
        Monitoring:
          MonitoredPV = ::AlarmMgr:Alarms[65]
          TriggerValues:
            [0] = 1
    [80]:
      Name = Alarm66
      Message = {$Alarms/Alarm.66}
      Code = 66
      Behavior = DiscreteValueMonitoring
        Monitoring:
          MonitoredPV = ::AlarmMgr:Alarms[66]
          TriggerValues:
            [0] = 1
    [81]:
      Name = Alarm67
      Message = {$Alarms/Alarm.67}
      Code = 67
      Behavior = DiscreteValueMonitoring
        Monitoring:
          MonitoredPV = ::AlarmMgr:Alarms[67]
          TriggerValues:
            [0] = 1
    [82]:
      Name = Alarm68
      Message = {$Alarms/Alarm.68}
      Code = 68
      Behavior = DiscreteValueMonitoring
        Monitoring:
          MonitoredPV = ::AlarmMgr:Alarms[68]
          TriggerValues:
            [0] = 1
    [83]:
      Name = Alarm69
      Message = {$Alarms/Alarm.69}
      Code = 69
      Behavior = DiscreteValueMonitoring
        Monitoring:
          MonitoredPV = ::AlarmMgr:Alarms[69]
          TriggerValues:
            [0] = 1
    [84]:
      Name = Alarm70
      Message = {$Alarms/Alarm.70}
      Behavior = DiscreteValueMonitoring
        Monitoring:
          MonitoredPV = ::AlarmMgr:Alarms[70]
          TriggerValues:
            [0] = 1
    [85]:
      Name = Alarm71
      Message = {$Alarms/Alarm.71}
      Code = 71
      Behavior = DiscreteValueMonitoring
        Monitoring:
          MonitoredPV = ::AlarmMgr:Alarms[71]
          TriggerValues:
            [0] = 1
    [86]:
      Name = Alarm72
      Message = {$Alarms/Alarm.72}
      Code = 72
      Behavior = DiscreteValueMonitoring
        Monitoring:
          MonitoredPV = ::AlarmMgr:Alarms[72]
          TriggerValues:
            [0] = 1
    [87]:
      Name = Alarm73
      Message = {$Alarms/Alarm.73}
      Code = 73
      Behavior = DiscreteValueMonitoring
        Monitoring:
          MonitoredPV = ::AlarmMgr:Alarms[73]
          TriggerValues:
            [0] = 1
    [88]:
      Name = Alarm74
      Message = {$Alarms/Alarm.74}
      Code = 74
      Behavior = DiscreteValueMonitoring
        Monitoring:
          MonitoredPV = ::AlarmMgr:Alarms[74]
          TriggerValues:
            [0] = 1
    [89]:
      Name = Alarm75
      Message = {$Alarms/Alarm.75}
      Code = 75
      Behavior = DiscreteValueMonitoring
        Monitoring:
          MonitoredPV = ::AlarmMgr:Alarms[75]
          TriggerValues:
            [0] = 1
    [90]:
      Name = Alarm76
      Message = {$Alarms/Alarm.76}
      Code = 76
      Behavior = DiscreteValueMonitoring
        Monitoring:
          MonitoredPV = ::AlarmMgr:Alarms[76]
          TriggerValues:
            [0] = 1
    [91]:
      Name = Alarm77
      Message = {$Alarms/Alarm.77}
      Code = 77
      Behavior = DiscreteValueMonitoring
        Monitoring:
          MonitoredPV = ::AlarmMgr:Alarms[77]
          TriggerValues:
            [0] = 1
    [92]:
      Name = Alarm78
      Message = {$Alarms/Alarm.78}
      Code = 78
      Behavior = DiscreteValueMonitoring
        Monitoring:
          MonitoredPV = ::AlarmMgr:Alarms[78]
          TriggerValues:
            [0] = 1
    [93]:
      Name = Alarm79
      Message = {$Alarms/Alarm.79}
      Code = 79
      Behavior = DiscreteValueMonitoring
        Monitoring:
          MonitoredPV = ::AlarmMgr:Alarms[79]
          TriggerValues:
            [0] = 1
    [94]:
      Name = Alarm80
      Message = {$Alarms/Alarm.80}
      Behavior = DiscreteValueMonitoring
        Monitoring:
          MonitoredPV = ::AlarmMgr:Alarms[80]
          TriggerValues:
            [0] = 1
    [95]:
      Name = Alarm81
      Message = {$Alarms/Alarm.81}
      Code = 81
      Behavior = DiscreteValueMonitoring
        Monitoring:
          MonitoredPV = ::AlarmMgr:Alarms[81]
          TriggerValues:
            [0] = 1
    [96]:
      Name = Alarm82
      Message = {$Alarms/Alarm.82}
      Code = 82
      Behavior = DiscreteValueMonitoring
        Monitoring:
          MonitoredPV = ::AlarmMgr:Alarms[82]
          TriggerValues:
            [0] = 1
    [97]:
      Name = Alarm83
      Message = {$Alarms/Alarm.83}
      Code = 83
      Behavior = DiscreteValueMonitoring
        Monitoring:
          MonitoredPV = ::AlarmMgr:Alarms[83]
          TriggerValues:
            [0] = 1
    [98]:
      Name = Alarm84
      Message = {$Alarms/Alarm.84}
      Code = 84
      Behavior = DiscreteValueMonitoring
        Monitoring:
          MonitoredPV = ::AlarmMgr:Alarms[84]
          TriggerValues:
            [0] = 1
    [99]:
      Name = Alarm85
      Message = {$Alarms/Alarm.85}
      Code = 85
      Behavior = DiscreteValueMonitoring
        Monitoring:
          MonitoredPV = ::AlarmMgr:Alarms[85]
          TriggerValues:
            [0] = 1
    [100]:
      Name = Alarm86
      Message = {$Alarms/Alarm.86}
      Code = 86
      Behavior = DiscreteValueMonitoring
        Monitoring:
          MonitoredPV = ::AlarmMgr:Alarms[86]
          TriggerValues:
            [0] = 1
    [101]:
      Name = Alarm87
      Message = {$Alarms/Alarm.87}
      Code = 87
      Behavior = DiscreteValueMonitoring
        Monitoring:
          MonitoredPV = ::AlarmMgr:Alarms[87]
          TriggerValues:
            [0] = 1
    [102]:
      Name = Alarm88
      Message = {$Alarms/Alarm.88}
      Code = 88
      Behavior = DiscreteValueMonitoring
        Monitoring:
          MonitoredPV = ::AlarmMgr:Alarms[88]
          TriggerValues:
            [0] = 1
    [103]:
      Name = Alarm89
      Message = {$Alarms/Alarm.89}
      Code = 89
      Behavior = DiscreteValueMonitoring
        Monitoring:
          MonitoredPV = ::AlarmMgr:Alarms[89]
          TriggerValues:
            [0] = 1
    [104]:
      Name = Alarm90
      Message = {$Alarms/Alarm.90}
      Behavior = DiscreteValueMonitoring
        Monitoring:
          MonitoredPV = ::AlarmMgr:Alarms[90]
          TriggerValues:
            [0] = 1
    [105]:
      Name = Alarm91
      Message = {$Alarms/Alarm.91}
      Code = 91
      Behavior = DiscreteValueMonitoring
        Monitoring:
          MonitoredPV = ::AlarmMgr:Alarms[91]
          TriggerValues:
            [0] = 1
    [106]:
      Name = Alarm92
      Message = {$Alarms/Alarm.92}
      Code = 92
      Behavior = DiscreteValueMonitoring
        Monitoring:
          MonitoredPV = ::AlarmMgr:Alarms[92]
          TriggerValues:
            [0] = 1
    [107]:
      Name = Alarm93
      Message = {$Alarms/Alarm.93}
      Code = 93
      Behavior = DiscreteValueMonitoring
        Monitoring:
          MonitoredPV = ::AlarmMgr:Alarms[93]
          TriggerValues:
            [0] = 1
    [108]:
      Name = Alarm94
      Message = {$Alarms/Alarm.94}
      Code = 94
      Behavior = DiscreteValueMonitoring
        Monitoring:
          MonitoredPV = ::AlarmMgr:Alarms[94]
          TriggerValues:
            [0] = 1
    [109]:
      Name = Alarm95
      Message = {$Alarms/Alarm.95}
      Code = 95
      Behavior = DiscreteValueMonitoring
        Monitoring:
          MonitoredPV = ::AlarmMgr:Alarms[95]
          TriggerValues:
            [0] = 1
    [110]:
      Name = Alarm96
      Message = {$Alarms/Alarm.96}
      Code = 96
      Behavior = DiscreteValueMonitoring
        Monitoring:
          MonitoredPV = ::AlarmMgr:Alarms[96]
          TriggerValues:
            [0] = 1
    [111]:
      Name = Alarm97
      Message = {$Alarms/Alarm.97}
      Code = 97
      Behavior = DiscreteValueMonitoring
        Monitoring:
          MonitoredPV = ::AlarmMgr:Alarms[97]
          TriggerValues:
            [0] = 1
    [112]:
      Name = Alarm98
      Message = {$Alarms/Alarm.98}
      Code = 98
      Behavior = DiscreteValueMonitoring
        Monitoring:
          MonitoredPV = ::AlarmMgr:Alarms[98]
          TriggerValues:
            [0] = 1
    [113]:
      Name = Alarm99
      Message = {$Alarms/Alarm.99}
      Code = 99
      Behavior = DiscreteValueMonitoring
        Monitoring:
          MonitoredPV = ::AlarmMgr:Alarms[99]
          TriggerValues:
            [0] = 1
  mapp.AlarmX.Core.Snippets:
    AutoDetect = 1
    [0]:
      Key = snippet1
      Value:
        PV = ::AlarmMgr:AlarmExamples.SnippetValue
  mapp.AlarmX.Core.Queries:
    [0]:
      Name = ActiveAlarms
      Update = ::AlarmMgr:AlarmQuery.UpdateCount
      Source:
        SELECT:
          [0]:
            PV = ::AlarmMgr:AlarmQuery.Alarms[].Name
          [1]:
            Column = Message
            PV = ::AlarmMgr:AlarmQuery.Alarms[].Message
          [2]:
            Column = Code
            PV = ::AlarmMgr:AlarmQuery.Alarms[].Code
          [3]:
            Column = Severity
            PV = ::AlarmMgr:AlarmQuery.Alarms[].Severity
          [4]:
            Column = Scope
            PV = ::AlarmMgr:AlarmQuery.Alarms[].Scope
          [5]:
            Column = TimeStamp
            PV = ::AlarmMgr:AlarmQuery.Alarms[].TimeStamp
          [6]:
            Column = AdditionalInformation1
            PV = ::AlarmMgr:AlarmQuery.Alarms[].AdditionalInfo
          [7]:
            Column = StateActive
            PV = ::AlarmMgr:AlarmQuery.Alarms[].Active
          [8]:
            Column = StateAcknowledged
            PV = ::AlarmMgr:AlarmQuery.Alarms[].Acknowledged
```

### AlmHistory.mpalarmxhistory - 5PPC2200_AL14_000/mappServices/AlarmX/AlmHistory.mpalarmxhistory
```
Element gAlarmXHistoryMpLink (Type=mpalarmxhistory)
  mapp.AlarmX.History:
    Memory:
      MemorySize = 6000
    Auditing = MpAudit
    Scope = Branch
```
